// TIA Portal V20 export
FUNCTION_BLOCK "Sequence_10_GuageRnR"   // FB224, LAD
TITLE = Sequence
// Sequence template programmend in ladder logic
// stored: IsIECCheckEnabled true, MemoryReserve 100, Namespace Unit1.Em8, SetENOAutomatically true
   VAR_INPUT
      unitStatus { ExternalAccessible := 'False'; ExternalVisible := 'False'; ExternalWritable := 'False'} : "LAF_typeUnitStatus";
   END_VAR
   VAR
      instSequenceLADControl { ExternalAccessible := 'False'; ExternalVisible := 'False'; ExternalWritable := 'False'} : "LAF_ControlLadSequence";
      instSequenceLADStatus { ExternalAccessible := 'False'; ExternalVisible := 'False'; ExternalWritable := 'False'} : "LAF_StatusLadSequence";
      statTonTime { ExternalAccessible := 'False'; ExternalVisible := 'False'; ExternalWritable := 'False'} : Array[0..9999] of TON_TIME;
      NoDataCheck { S7_SetPoint := 'True'} : "LER_typePartData";
   END_VAR
   VAR_TEMP
      tempCustomerAction : Bool;   // Placeholder for possible actions
      tempDo_nothing_and_wait_for_init : Bool;   // Placeholder for doing nothing
      tempSafeStateCondition : Bool;   // Temp Condition for the equipment module to be in a safe state
   END_VAR
   VAR CONSTANT
      delayTime : Time := T#500ms;
      STEP_IDLE : DInt := 1;
      JOB_1_STEP_01 : DInt := 101;
      JOB_1_STEP_10 : DInt := 110;
      JOB_1_STEP_11 : DInt := 111;
      JOB_1_STEP_20 : DInt := 120;
      JOB_1_STEP_21 : DInt := 121;
      JOB_1_STEP_30 : DInt := 130;
      JOB_1_STEP_40 : DInt := 140;
      JOB_1_STEP_41 : DInt := 141;
      JOB_1_STEP_50 : DInt := 150;
      JOB_1_STEP_60 : DInt := 160;
      JOB_1_STEP_70 : DInt := 170;
      JOB_1_STEP_80 : DInt := 180;
      JOB_1_STEP_90 : DInt := 190;
      JOB_2_STEP_01 : DInt := 201;
      JOB_2_STEP_10 : DInt := 210;
      JOB_2_STEP_20 : DInt := 220;
      JOB_2_STEP_30 : DInt := 230;
      JOB_2_STEP_31 : DInt := 231;
      JOB_2_STEP_32 : DInt := 232;
      JOB_2_STEP_40 : DInt := 240;
      JOB_2_STEP_41 : DInt := 241;
      JOB_2_STEP_42 : DInt := 242;
      JOB_2_STEP_43 : DInt := 242;
      JOB_2_STEP_50 : DInt := 250;
      JOB_2_STEP_60 : DInt := 260;
      JOB_2_STEP_70 : DInt := 270;
      JOB_2_STEP_80 : DInt := 280;
      JOB_2_STEP_90 : DInt := 290;
      JOB_3_STEP_01 : DInt := 301;
      JOB_3_STEP_10 : DInt := 310;
      JOB_3_STEP_11 : DInt := 311;
      JOB_3_STEP_20 : DInt := 320;
      JOB_3_STEP_30 : DInt := 330;
      JOB_3_STEP_31 : DInt := 331;
      JOB_3_STEP_32 : DInt := 332;
      JOB_3_STEP_33 : DInt := 333;
      JOB_3_STEP_34 : DInt := 334;
      JOB_3_STEP_35 : DInt := 335;
      JOB_3_STEP_36 : DInt := 336;
      JOB_3_STEP_37 : DInt := 337;
      JOB_3_STEP_38 : DInt := 338;
      JOB_3_STEP_40 : DInt := 340;
      JOB_3_STEP_45 : DInt := 345;
      JOB_3_STEP_50 : DInt := 350;
      JOB_3_STEP_51 : DInt := 351;
      JOB_3_STEP_52 : DInt := 352;
      JOB_3_STEP_60 : DInt := 360;
      JOB_3_STEP_61 : DInt := 361;
      JOB_3_STEP_62 : DInt := 362;
      JOB_3_STEP_63 : DInt := 363;
      JOB_3_STEP_70 : DInt := 370;
      JOB_3_STEP_80 : DInt := 380;
      JOB_3_STEP_90 : DInt := 390;
      JOB_4_STEP_01 : DInt := 401;
      JOB_4_STEP_10 : DInt := 410;
      JOB_4_STEP_20 : DInt := 420;
      JOB_4_STEP_30 : DInt := 430;
      JOB_4_STEP_31 : DInt := 431;
      JOB_4_STEP_40 : DInt := 440;
      JOB_4_STEP_41 : DInt := 441;
      JOB_4_STEP_42 : DInt := 442;
      JOB_4_STEP_50 : DInt := 450;
      JOB_4_STEP_60 : DInt := 460;
      JOB_4_STEP_70 : DInt := 470;
      JOB_4_STEP_80 : DInt := 480;
      JOB_4_STEP_81 : DInt := 481;
      JOB_4_STEP_90 : DInt := 490;
      JOB_5_STEP_01 : DInt := 501;
      JOB_5_STEP_10 : DInt := 510;
      JOB_5_STEP_11 : DInt := 511;
      JOB_5_STEP_12 : DInt := 512;
      JOB_5_STEP_13 : DInt := 513;
      JOB_5_STEP_20 : DInt := 520;
      JOB_5_STEP_30 : DInt := 530;
      JOB_5_STEP_40 : DInt := 540;
      JOB_5_STEP_41 : DInt := 541;
      JOB_5_STEP_42 : DInt := 542;
      JOB_5_STEP_43 : DInt := 543;
      JOB_5_STEP_44 : DInt := 544;
      JOB_5_STEP_45 : DInt := 545;
      JOB_5_STEP_46 : DInt := 546;
      JOB_5_STEP_47 : DInt := 547;
      JOB_5_STEP_48 : DInt := 548;
      JOB_5_STEP_50 : DInt := 550;
      JOB_5_STEP_60 : DInt := 560;
      JOB_5_STEP_61 : DInt := 561;
      JOB_5_STEP_62 : DInt := 562;
      JOB_5_STEP_63 : DInt := 563;
      JOB_5_STEP_64 : DInt := 564;
      STEP_IMMEDIATE_STOP : DInt := 9001;   // Step executed when an immediate stop command is triggered for the sequence (i.e. when unit is in state aborting)
   END_VAR
   VAR_TEMP   // added for the SCL form of the ladder/FBD networks
      _w1 : Bool;
      _w2 : Bool;
      _w3 : Bool;
   END_VAR
BEGIN

REGION Network 1: BLOCK INFO HEADER
   // (company) / (C) Copyright (year)
   // ---------------------------------------------------------------------------------
   // Title:                             (Title of this block)
   // Comment/Function: (that is implemented in the block)
   // Library/Family:           (that the source is dedicated to)
   // Author:                        (department / person in charge / contact)
   // Target System:          (test system with FW version)
   // Engineering:              TIA Portal (SW version)
   // Restrictions:               (OB types, etc.)
   // Requirements:           (hardware, technological package, etc.)
   // ---------------------------------------------------------------------------------
   // Change log table:
   // Version          | Date             | Signature      | Expert in charge  | Changes applied ------------------------|----------------------|-------------------------|--------------------------------|-----------------------
   // 001.000.000 | yyyy-mm-dd | 0x00000000 | (name of expert) | First released version
END_REGION

REGION Network 2: DESCRIPTION
   // This is a template block provided by the Automation Framework. It can be used to create an own project.
   // The Block Info Header is prepared to put in your own data.
   // Description of the block could be added here and the docu created by Code2Docu.
END_REGION

REGION Network 3: ********************* CONTROL *************************
END_REGION

REGION Network 4: Sequence Control ("Enter your Sequins number here")
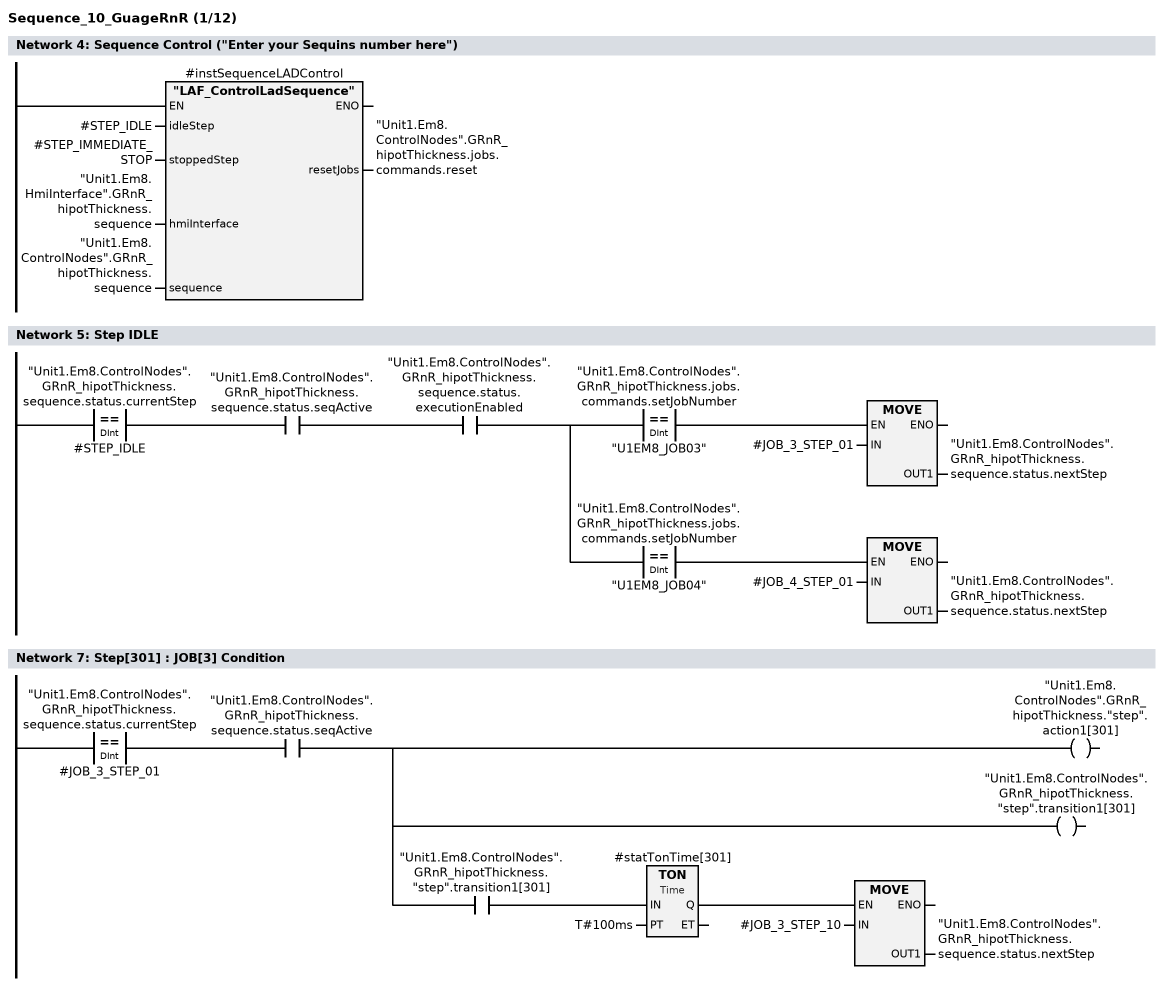
   RUNG wire#powerrail
      #instSequenceLADControl(idleStep := #STEP_IDLE, stoppedStep := #STEP_IMMEDIATE_STOP, hmiInterface := "Unit1.Em8.HmiInterface".GRnR_hipotThickness.sequence, sequence := "Unit1.Em8.ControlNodes".GRnR_hipotThickness.sequence, resetJobs => "Unit1.Em8.ControlNodes".GRnR_hipotThickness.jobs.commands.reset)
   END_RUNG
   // the same network as SCL:
   #instSequenceLADControl(idleStep := #STEP_IDLE,   // "LAF_ControlLadSequence"
                           stoppedStep := #STEP_IMMEDIATE_STOP,
                           hmiInterface := "Unit1.Em8.HmiInterface".GRnR_hipotThickness.sequence,
                           sequence := "Unit1.Em8.ControlNodes".GRnR_hipotThickness.sequence,
                           resetJobs => "Unit1.Em8.ControlNodes".GRnR_hipotThickness.jobs.commands.reset);
END_REGION

REGION Network 5: Step IDLE
   RUNG wire#powerrail
      { S7_Templates := "SrcType := DInt" } EQ_Contact(in1 := "Unit1.Em8.ControlNodes".GRnR_hipotThickness.sequence.status.currentStep, in2 := #STEP_IDLE)
      Contact( "Unit1.Em8.ControlNodes".GRnR_hipotThickness.sequence.status.seqActive )
      Contact( "Unit1.Em8.ControlNodes".GRnR_hipotThickness.sequence.status.executionEnabled )
      wire#w1
      { S7_Templates := "SrcType := DInt" } EQ_Contact(in1 := "Unit1.Em8.ControlNodes".GRnR_hipotThickness.jobs.commands.setJobNumber, in2 := "U1EM8_JOB03")
      Move(in := #JOB_3_STEP_01, out1 => "Unit1.Em8.ControlNodes".GRnR_hipotThickness.sequence.status.nextStep)
   END_RUNG
   RUNG wire#w1
      { S7_Templates := "SrcType := DInt" } EQ_Contact(in1 := "Unit1.Em8.ControlNodes".GRnR_hipotThickness.jobs.commands.setJobNumber, in2 := "U1EM8_JOB04")
      Move(in := #JOB_4_STEP_01, out1 => "Unit1.Em8.ControlNodes".GRnR_hipotThickness.sequence.status.nextStep)
   END_RUNG
   // the same network as SCL:
   #_w1 := ("Unit1.Em8.ControlNodes".GRnR_hipotThickness.sequence.status.currentStep = #STEP_IDLE) AND "Unit1.Em8.ControlNodes".GRnR_hipotThickness.sequence.status.seqActive AND "Unit1.Em8.ControlNodes".GRnR_hipotThickness.sequence.status.executionEnabled;
   IF #_w1 AND ("Unit1.Em8.ControlNodes".GRnR_hipotThickness.jobs.commands.setJobNumber = "U1EM8_JOB03") THEN
       "Unit1.Em8.ControlNodes".GRnR_hipotThickness.sequence.status.nextStep := #JOB_3_STEP_01;
   END_IF;
   IF #_w1 AND ("Unit1.Em8.ControlNodes".GRnR_hipotThickness.jobs.commands.setJobNumber = "U1EM8_JOB04") THEN
       "Unit1.Em8.ControlNodes".GRnR_hipotThickness.sequence.status.nextStep := #JOB_4_STEP_01;
   END_IF;
END_REGION

REGION Network 6: ************ JOB[3] JR HIPOT & THICKNESS=AUTO *************
END_REGION

REGION Network 7: Step[301] : JOB[3] Condition
   RUNG wire#powerrail
      { S7_Templates := "SrcType := DInt" } EQ_Contact(in1 := "Unit1.Em8.ControlNodes".GRnR_hipotThickness.sequence.status.currentStep, in2 := #JOB_3_STEP_01)
      Contact( "Unit1.Em8.ControlNodes".GRnR_hipotThickness.sequence.status.seqActive )
      wire#w1
      Coil( "Unit1.Em8.ControlNodes".GRnR_hipotThickness."step".action1[301] )
   END_RUNG
   RUNG wire#w1
      Coil( "Unit1.Em8.ControlNodes".GRnR_hipotThickness."step".transition1[301] )
   END_RUNG
   RUNG wire#w1
      Contact( "Unit1.Em8.ControlNodes".GRnR_hipotThickness."step".transition1[301] )
      { S7_Templates := "time_type := Time" } #statTonTime[301].TON(pt := T#100ms, et =>)
      Move(in := #JOB_3_STEP_10, out1 => "Unit1.Em8.ControlNodes".GRnR_hipotThickness.sequence.status.nextStep)
   END_RUNG
   // the same network as SCL:
   "Unit1.Em8.ControlNodes".GRnR_hipotThickness."step".action1[301] := ("Unit1.Em8.ControlNodes".GRnR_hipotThickness.sequence.status.currentStep = #JOB_3_STEP_01) AND "Unit1.Em8.ControlNodes".GRnR_hipotThickness.sequence.status.seqActive;
   "Unit1.Em8.ControlNodes".GRnR_hipotThickness."step".transition1[301] := ("Unit1.Em8.ControlNodes".GRnR_hipotThickness.sequence.status.currentStep = #JOB_3_STEP_01) AND "Unit1.Em8.ControlNodes".GRnR_hipotThickness.sequence.status.seqActive;
   #statTonTime[301].TON(IN := ("Unit1.Em8.ControlNodes".GRnR_hipotThickness.sequence.status.currentStep = #JOB_3_STEP_01) AND "Unit1.Em8.ControlNodes".GRnR_hipotThickness.sequence.status.seqActive AND "Unit1.Em8.ControlNodes".GRnR_hipotThickness."step".transition1[301],
                         PT := T#100ms);
   IF #statTonTime[301].Q THEN
       "Unit1.Em8.ControlNodes".GRnR_hipotThickness.sequence.status.nextStep := #JOB_3_STEP_10;
   END_IF;
END_REGION

REGION Network 8: Step[310] : Stage Lift Down
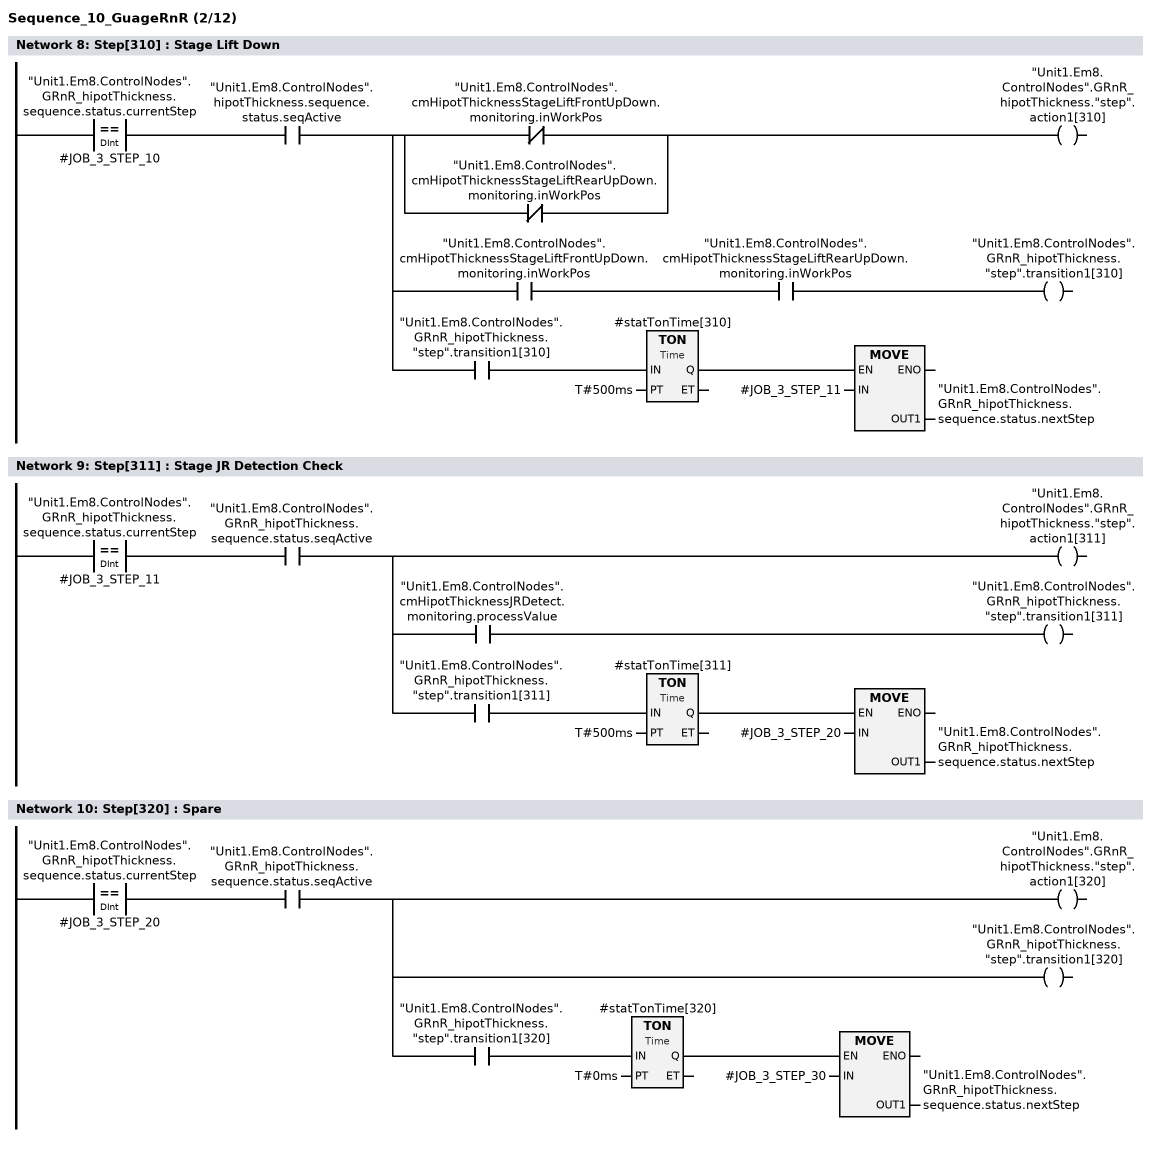
   RUNG wire#powerrail
      { S7_Templates := "SrcType := DInt" } EQ_Contact(in1 := "Unit1.Em8.ControlNodes".GRnR_hipotThickness.sequence.status.currentStep, in2 := #JOB_3_STEP_10)
      Contact( "Unit1.Em8.ControlNodes".hipotThickness.sequence.status.seqActive )
      wire#w1
      I_Contact( "Unit1.Em8.ControlNodes".cmHipotThicknessStageLiftFrontUpDown.monitoring.inWorkPos )
      wire#w2
      Coil( "Unit1.Em8.ControlNodes".GRnR_hipotThickness."step".action1[310] )
   END_RUNG
   RUNG wire#w1
      I_Contact( "Unit1.Em8.ControlNodes".cmHipotThicknessStageLiftRearUpDown.monitoring.inWorkPos )
   END_RUNG wire#w2
   RUNG wire#w1
      Contact( "Unit1.Em8.ControlNodes".cmHipotThicknessStageLiftFrontUpDown.monitoring.inWorkPos )
      Contact( "Unit1.Em8.ControlNodes".cmHipotThicknessStageLiftRearUpDown.monitoring.inWorkPos )
      Coil( "Unit1.Em8.ControlNodes".GRnR_hipotThickness."step".transition1[310] )
   END_RUNG
   RUNG wire#w1
      Contact( "Unit1.Em8.ControlNodes".GRnR_hipotThickness."step".transition1[310] )
      { S7_Templates := "time_type := Time" } #statTonTime[310].TON(pt := T#500ms, et =>)
      Move(in := #JOB_3_STEP_11, out1 => "Unit1.Em8.ControlNodes".GRnR_hipotThickness.sequence.status.nextStep)
   END_RUNG
   // the same network as SCL:
   #_w1 := ("Unit1.Em8.ControlNodes".GRnR_hipotThickness.sequence.status.currentStep = #JOB_3_STEP_10) AND "Unit1.Em8.ControlNodes".hipotThickness.sequence.status.seqActive;
   "Unit1.Em8.ControlNodes".GRnR_hipotThickness."step".action1[310] := #_w1 AND (NOT "Unit1.Em8.ControlNodes".cmHipotThicknessStageLiftFrontUpDown.monitoring.inWorkPos OR NOT "Unit1.Em8.ControlNodes".cmHipotThicknessStageLiftRearUpDown.monitoring.inWorkPos);
   "Unit1.Em8.ControlNodes".GRnR_hipotThickness."step".transition1[310] := #_w1 AND "Unit1.Em8.ControlNodes".cmHipotThicknessStageLiftFrontUpDown.monitoring.inWorkPos AND "Unit1.Em8.ControlNodes".cmHipotThicknessStageLiftRearUpDown.monitoring.inWorkPos;
   #statTonTime[310].TON(IN := #_w1 AND "Unit1.Em8.ControlNodes".GRnR_hipotThickness."step".transition1[310],
                         PT := T#500ms);
   IF #statTonTime[310].Q THEN
       "Unit1.Em8.ControlNodes".GRnR_hipotThickness.sequence.status.nextStep := #JOB_3_STEP_11;
   END_IF;
END_REGION

REGION Network 9: Step[311] : Stage JR Detection Check
   RUNG wire#powerrail
      { S7_Templates := "SrcType := DInt" } EQ_Contact(in1 := "Unit1.Em8.ControlNodes".GRnR_hipotThickness.sequence.status.currentStep, in2 := #JOB_3_STEP_11)
      Contact( "Unit1.Em8.ControlNodes".GRnR_hipotThickness.sequence.status.seqActive )
      wire#w1
      Coil( "Unit1.Em8.ControlNodes".GRnR_hipotThickness."step".action1[311] )
   END_RUNG
   RUNG wire#w1
      Contact( "Unit1.Em8.ControlNodes".cmHipotThicknessJRDetect.monitoring.processValue )
      Coil( "Unit1.Em8.ControlNodes".GRnR_hipotThickness."step".transition1[311] )
   END_RUNG
   RUNG wire#w1
      Contact( "Unit1.Em8.ControlNodes".GRnR_hipotThickness."step".transition1[311] )
      { S7_Templates := "time_type := Time" } #statTonTime[311].TON(pt := T#500ms, et =>)
      Move(in := #JOB_3_STEP_20, out1 => "Unit1.Em8.ControlNodes".GRnR_hipotThickness.sequence.status.nextStep)
   END_RUNG
   // the same network as SCL:
   "Unit1.Em8.ControlNodes".GRnR_hipotThickness."step".action1[311] := ("Unit1.Em8.ControlNodes".GRnR_hipotThickness.sequence.status.currentStep = #JOB_3_STEP_11) AND "Unit1.Em8.ControlNodes".GRnR_hipotThickness.sequence.status.seqActive;
   "Unit1.Em8.ControlNodes".GRnR_hipotThickness."step".transition1[311] := ("Unit1.Em8.ControlNodes".GRnR_hipotThickness.sequence.status.currentStep = #JOB_3_STEP_11) AND "Unit1.Em8.ControlNodes".GRnR_hipotThickness.sequence.status.seqActive AND "Unit1.Em8.ControlNodes".cmHipotThicknessJRDetect.monitoring.processValue;
   #statTonTime[311].TON(IN := ("Unit1.Em8.ControlNodes".GRnR_hipotThickness.sequence.status.currentStep = #JOB_3_STEP_11) AND "Unit1.Em8.ControlNodes".GRnR_hipotThickness.sequence.status.seqActive AND "Unit1.Em8.ControlNodes".GRnR_hipotThickness."step".transition1[311],
                         PT := T#500ms);
   IF #statTonTime[311].Q THEN
       "Unit1.Em8.ControlNodes".GRnR_hipotThickness.sequence.status.nextStep := #JOB_3_STEP_20;
   END_IF;
END_REGION

REGION Network 10: Step[320] : Spare
   RUNG wire#powerrail
      { S7_Templates := "SrcType := DInt" } EQ_Contact(in1 := "Unit1.Em8.ControlNodes".GRnR_hipotThickness.sequence.status.currentStep, in2 := #JOB_3_STEP_20)
      Contact( "Unit1.Em8.ControlNodes".GRnR_hipotThickness.sequence.status.seqActive )
      wire#w1
      Coil( "Unit1.Em8.ControlNodes".GRnR_hipotThickness."step".action1[320] )
   END_RUNG
   RUNG wire#w1
      Coil( "Unit1.Em8.ControlNodes".GRnR_hipotThickness."step".transition1[320] )
   END_RUNG
   RUNG wire#w1
      Contact( "Unit1.Em8.ControlNodes".GRnR_hipotThickness."step".transition1[320] )
      { S7_Templates := "time_type := Time" } #statTonTime[320].TON(pt := T#0ms, et =>)
      Move(in := #JOB_3_STEP_30, out1 => "Unit1.Em8.ControlNodes".GRnR_hipotThickness.sequence.status.nextStep)
   END_RUNG
   // the same network as SCL:
   "Unit1.Em8.ControlNodes".GRnR_hipotThickness."step".action1[320] := ("Unit1.Em8.ControlNodes".GRnR_hipotThickness.sequence.status.currentStep = #JOB_3_STEP_20) AND "Unit1.Em8.ControlNodes".GRnR_hipotThickness.sequence.status.seqActive;
   "Unit1.Em8.ControlNodes".GRnR_hipotThickness."step".transition1[320] := ("Unit1.Em8.ControlNodes".GRnR_hipotThickness.sequence.status.currentStep = #JOB_3_STEP_20) AND "Unit1.Em8.ControlNodes".GRnR_hipotThickness.sequence.status.seqActive;
   #statTonTime[320].TON(IN := ("Unit1.Em8.ControlNodes".GRnR_hipotThickness.sequence.status.currentStep = #JOB_3_STEP_20) AND "Unit1.Em8.ControlNodes".GRnR_hipotThickness.sequence.status.seqActive AND "Unit1.Em8.ControlNodes".GRnR_hipotThickness."step".transition1[320],
                         PT := T#0ms);
   IF #statTonTime[320].Q THEN
       "Unit1.Em8.ControlNodes".GRnR_hipotThickness.sequence.status.nextStep := #JOB_3_STEP_30;
   END_IF;
END_REGION

REGION Network 11: Step[330] : Press Start
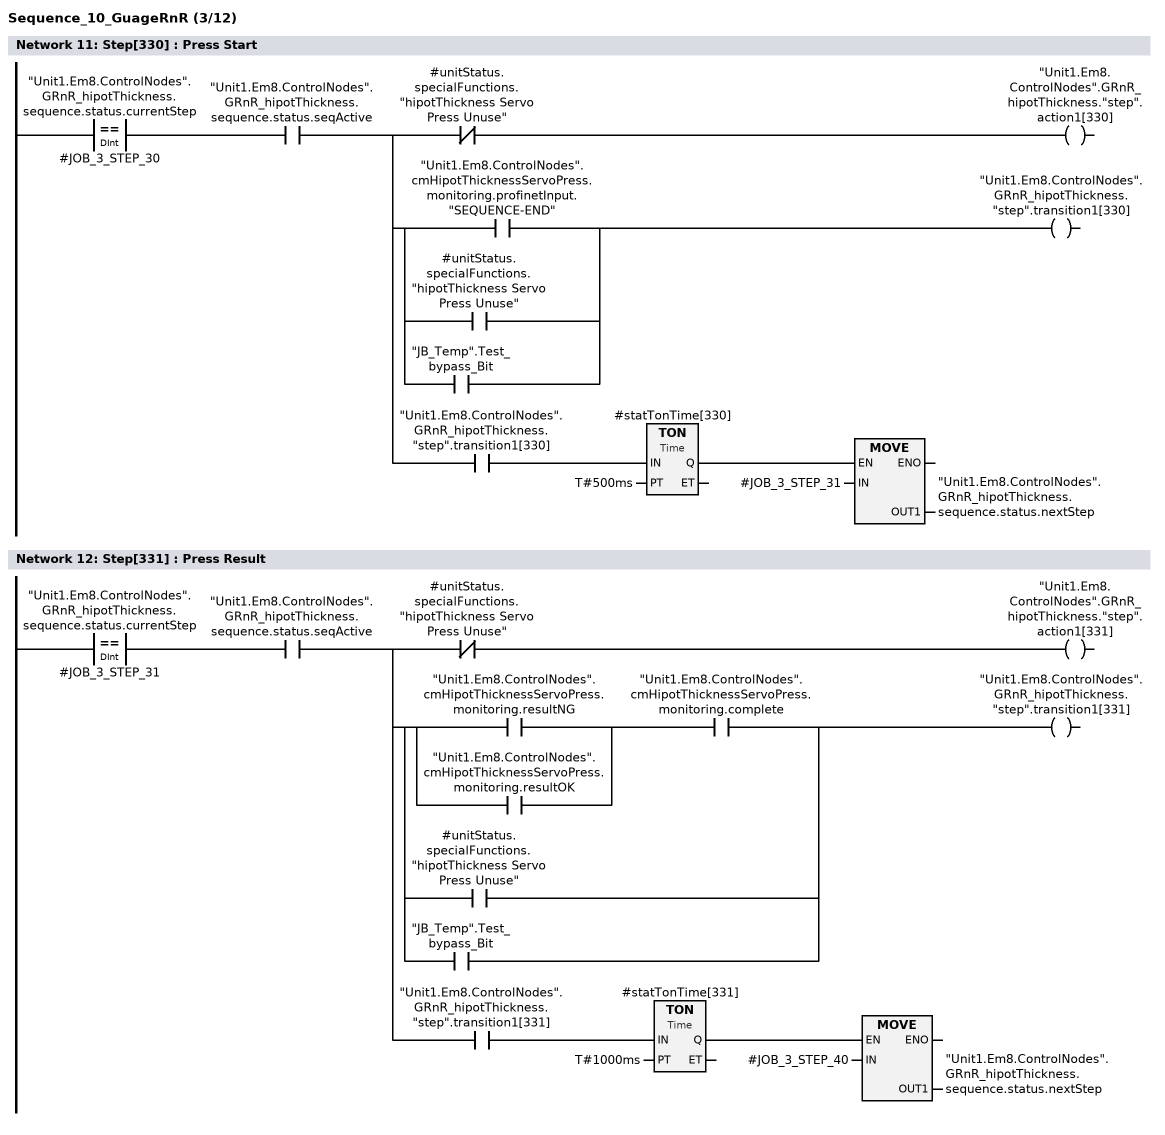
   RUNG wire#powerrail
      { S7_Templates := "SrcType := DInt" } EQ_Contact(in1 := "Unit1.Em8.ControlNodes".GRnR_hipotThickness.sequence.status.currentStep, in2 := #JOB_3_STEP_30)
      Contact( "Unit1.Em8.ControlNodes".GRnR_hipotThickness.sequence.status.seqActive )
      wire#w1
      I_Contact( #unitStatus.specialFunctions."hipotThickness Servo Press Unuse" )
      Coil( "Unit1.Em8.ControlNodes".GRnR_hipotThickness."step".action1[330] )
   END_RUNG
   RUNG wire#w1
      Contact( "Unit1.Em8.ControlNodes".cmHipotThicknessServoPress.monitoring.profinetInput."SEQUENCE-END" )
      wire#w2
      Coil( "Unit1.Em8.ControlNodes".GRnR_hipotThickness."step".transition1[330] )
   END_RUNG
   RUNG wire#w1
      Contact( #unitStatus.specialFunctions."hipotThickness Servo Press Unuse" )
   END_RUNG wire#w2
   RUNG wire#w1
      Contact( "JB_Temp".Test_bypass_Bit )
   END_RUNG wire#w2
   RUNG wire#w1
      Contact( "Unit1.Em8.ControlNodes".GRnR_hipotThickness."step".transition1[330] )
      { S7_Templates := "time_type := Time" } #statTonTime[330].TON(pt := T#500ms, et =>)
      Move(in := #JOB_3_STEP_31, out1 => "Unit1.Em8.ControlNodes".GRnR_hipotThickness.sequence.status.nextStep)
   END_RUNG
   // the same network as SCL:
   #_w1 := ("Unit1.Em8.ControlNodes".GRnR_hipotThickness.sequence.status.currentStep = #JOB_3_STEP_30) AND "Unit1.Em8.ControlNodes".GRnR_hipotThickness.sequence.status.seqActive;
   "Unit1.Em8.ControlNodes".GRnR_hipotThickness."step".action1[330] := #_w1 AND NOT #unitStatus.specialFunctions."hipotThickness Servo Press Unuse";
   "Unit1.Em8.ControlNodes".GRnR_hipotThickness."step".transition1[330] := #_w1 AND ("Unit1.Em8.ControlNodes".cmHipotThicknessServoPress.monitoring.profinetInput."SEQUENCE-END" OR #unitStatus.specialFunctions."hipotThickness Servo Press Unuse" OR "JB_Temp".Test_bypass_Bit);
   #statTonTime[330].TON(IN := #_w1 AND "Unit1.Em8.ControlNodes".GRnR_hipotThickness."step".transition1[330],
                         PT := T#500ms);
   IF #statTonTime[330].Q THEN
       "Unit1.Em8.ControlNodes".GRnR_hipotThickness.sequence.status.nextStep := #JOB_3_STEP_31;
   END_IF;
END_REGION

REGION Network 12: Step[331] : Press Result
   RUNG wire#powerrail
      { S7_Templates := "SrcType := DInt" } EQ_Contact(in1 := "Unit1.Em8.ControlNodes".GRnR_hipotThickness.sequence.status.currentStep, in2 := #JOB_3_STEP_31)
      Contact( "Unit1.Em8.ControlNodes".GRnR_hipotThickness.sequence.status.seqActive )
      wire#w1
      I_Contact( #unitStatus.specialFunctions."hipotThickness Servo Press Unuse" )
      Coil( "Unit1.Em8.ControlNodes".GRnR_hipotThickness."step".action1[331] )
   END_RUNG
   RUNG wire#w1
      Contact( "Unit1.Em8.ControlNodes".cmHipotThicknessServoPress.monitoring.resultNG )
      wire#w2
      Contact( "Unit1.Em8.ControlNodes".cmHipotThicknessServoPress.monitoring.complete )
      wire#w3
      Coil( "Unit1.Em8.ControlNodes".GRnR_hipotThickness."step".transition1[331] )
   END_RUNG
   RUNG wire#w1
      Contact( "Unit1.Em8.ControlNodes".cmHipotThicknessServoPress.monitoring.resultOK )
   END_RUNG wire#w2
   RUNG wire#w1
      Contact( #unitStatus.specialFunctions."hipotThickness Servo Press Unuse" )
   END_RUNG wire#w3
   RUNG wire#w1
      Contact( "JB_Temp".Test_bypass_Bit )
   END_RUNG wire#w3
   RUNG wire#w1
      Contact( "Unit1.Em8.ControlNodes".GRnR_hipotThickness."step".transition1[331] )
      { S7_Templates := "time_type := Time" } #statTonTime[331].TON(pt := T#1000ms, et =>)
      Move(in := #JOB_3_STEP_40, out1 => "Unit1.Em8.ControlNodes".GRnR_hipotThickness.sequence.status.nextStep)
   END_RUNG
   // the same network as SCL:
   #_w1 := ("Unit1.Em8.ControlNodes".GRnR_hipotThickness.sequence.status.currentStep = #JOB_3_STEP_31) AND "Unit1.Em8.ControlNodes".GRnR_hipotThickness.sequence.status.seqActive;
   "Unit1.Em8.ControlNodes".GRnR_hipotThickness."step".action1[331] := #_w1 AND NOT #unitStatus.specialFunctions."hipotThickness Servo Press Unuse";
   "Unit1.Em8.ControlNodes".GRnR_hipotThickness."step".transition1[331] := #_w1 AND ((("Unit1.Em8.ControlNodes".cmHipotThicknessServoPress.monitoring.resultNG OR "Unit1.Em8.ControlNodes".cmHipotThicknessServoPress.monitoring.resultOK) AND "Unit1.Em8.ControlNodes".cmHipotThicknessServoPress.monitoring.complete) OR #unitStatus.specialFunctions."hipotThickness Servo Press Unuse" OR "JB_Temp".Test_bypass_Bit);
   #statTonTime[331].TON(IN := #_w1 AND "Unit1.Em8.ControlNodes".GRnR_hipotThickness."step".transition1[331],
                         PT := T#1000ms);
   IF #statTonTime[331].Q THEN
       "Unit1.Em8.ControlNodes".GRnR_hipotThickness.sequence.status.nextStep := #JOB_3_STEP_40;
   END_IF;
END_REGION

REGION Network 13: Step[340] : Thickness Z-Axis Thickness Ready Pos, Tab Forward
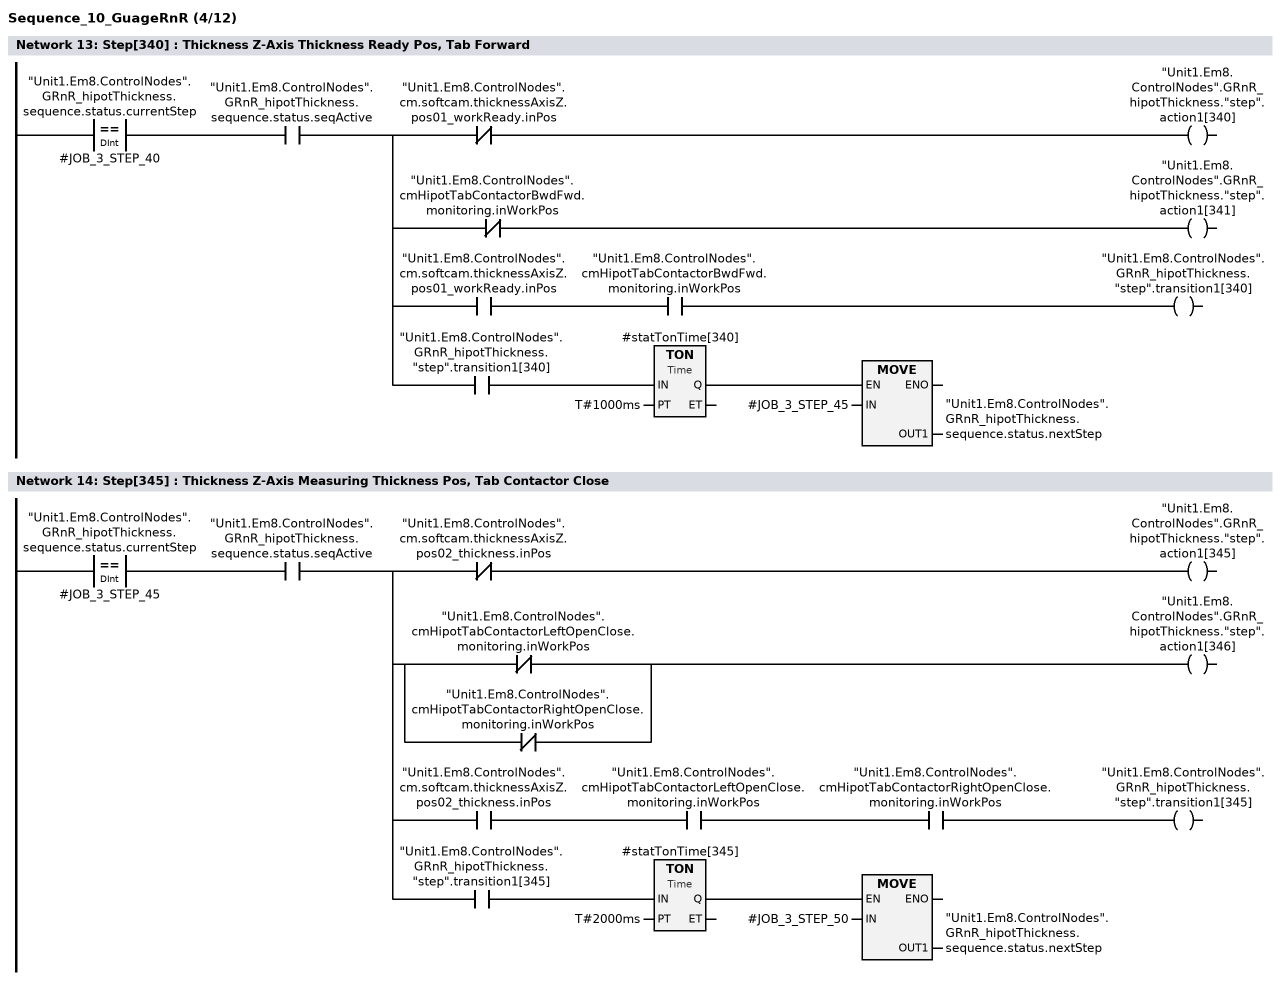
   RUNG wire#powerrail
      { S7_Templates := "SrcType := DInt" } EQ_Contact(in1 := "Unit1.Em8.ControlNodes".GRnR_hipotThickness.sequence.status.currentStep, in2 := #JOB_3_STEP_40)
      Contact( "Unit1.Em8.ControlNodes".GRnR_hipotThickness.sequence.status.seqActive )
      wire#w1
      I_Contact( "Unit1.Em8.ControlNodes".cm.softcam.thicknessAxisZ.pos01_workReady.inPos )
      Coil( "Unit1.Em8.ControlNodes".GRnR_hipotThickness."step".action1[340] )
   END_RUNG
   RUNG wire#w1
      I_Contact( "Unit1.Em8.ControlNodes".cmHipotTabContactorBwdFwd.monitoring.inWorkPos )
      Coil( "Unit1.Em8.ControlNodes".GRnR_hipotThickness."step".action1[341] )
   END_RUNG
   RUNG wire#w1
      Contact( "Unit1.Em8.ControlNodes".cm.softcam.thicknessAxisZ.pos01_workReady.inPos )
      Contact( "Unit1.Em8.ControlNodes".cmHipotTabContactorBwdFwd.monitoring.inWorkPos )
      Coil( "Unit1.Em8.ControlNodes".GRnR_hipotThickness."step".transition1[340] )
   END_RUNG
   RUNG wire#w1
      Contact( "Unit1.Em8.ControlNodes".GRnR_hipotThickness."step".transition1[340] )
      { S7_Templates := "time_type := Time" } #statTonTime[340].TON(pt := T#1000ms, et =>)
      Move(in := #JOB_3_STEP_45, out1 => "Unit1.Em8.ControlNodes".GRnR_hipotThickness.sequence.status.nextStep)
   END_RUNG
   // the same network as SCL:
   #_w1 := ("Unit1.Em8.ControlNodes".GRnR_hipotThickness.sequence.status.currentStep = #JOB_3_STEP_40) AND "Unit1.Em8.ControlNodes".GRnR_hipotThickness.sequence.status.seqActive;
   "Unit1.Em8.ControlNodes".GRnR_hipotThickness."step".action1[340] := #_w1 AND NOT "Unit1.Em8.ControlNodes".cm.softcam.thicknessAxisZ.pos01_workReady.inPos;
   "Unit1.Em8.ControlNodes".GRnR_hipotThickness."step".action1[341] := #_w1 AND NOT "Unit1.Em8.ControlNodes".cmHipotTabContactorBwdFwd.monitoring.inWorkPos;
   "Unit1.Em8.ControlNodes".GRnR_hipotThickness."step".transition1[340] := #_w1 AND "Unit1.Em8.ControlNodes".cm.softcam.thicknessAxisZ.pos01_workReady.inPos AND "Unit1.Em8.ControlNodes".cmHipotTabContactorBwdFwd.monitoring.inWorkPos;
   #statTonTime[340].TON(IN := #_w1 AND "Unit1.Em8.ControlNodes".GRnR_hipotThickness."step".transition1[340],
                         PT := T#1000ms);
   IF #statTonTime[340].Q THEN
       "Unit1.Em8.ControlNodes".GRnR_hipotThickness.sequence.status.nextStep := #JOB_3_STEP_45;
   END_IF;
END_REGION

REGION Network 14: Step[345] : Thickness Z-Axis Measuring Thickness Pos, Tab Contactor Close
   RUNG wire#powerrail
      { S7_Templates := "SrcType := DInt" } EQ_Contact(in1 := "Unit1.Em8.ControlNodes".GRnR_hipotThickness.sequence.status.currentStep, in2 := #JOB_3_STEP_45)
      Contact( "Unit1.Em8.ControlNodes".GRnR_hipotThickness.sequence.status.seqActive )
      wire#w1
      I_Contact( "Unit1.Em8.ControlNodes".cm.softcam.thicknessAxisZ.pos02_thickness.inPos )
      Coil( "Unit1.Em8.ControlNodes".GRnR_hipotThickness."step".action1[345] )
   END_RUNG
   RUNG wire#w1
      I_Contact( "Unit1.Em8.ControlNodes".cmHipotTabContactorLeftOpenClose.monitoring.inWorkPos )
      wire#w2
      Coil( "Unit1.Em8.ControlNodes".GRnR_hipotThickness."step".action1[346] )
   END_RUNG
   RUNG wire#w1
      I_Contact( "Unit1.Em8.ControlNodes".cmHipotTabContactorRightOpenClose.monitoring.inWorkPos )
   END_RUNG wire#w2
   RUNG wire#w1
      Contact( "Unit1.Em8.ControlNodes".cm.softcam.thicknessAxisZ.pos02_thickness.inPos )
      Contact( "Unit1.Em8.ControlNodes".cmHipotTabContactorLeftOpenClose.monitoring.inWorkPos )
      Contact( "Unit1.Em8.ControlNodes".cmHipotTabContactorRightOpenClose.monitoring.inWorkPos )
      Coil( "Unit1.Em8.ControlNodes".GRnR_hipotThickness."step".transition1[345] )
   END_RUNG
   RUNG wire#w1
      Contact( "Unit1.Em8.ControlNodes".GRnR_hipotThickness."step".transition1[345] )
      { S7_Templates := "time_type := Time" } #statTonTime[345].TON(pt := T#2000ms, et =>)
      Move(in := #JOB_3_STEP_50, out1 => "Unit1.Em8.ControlNodes".GRnR_hipotThickness.sequence.status.nextStep)
   END_RUNG
   // the same network as SCL:
   #_w1 := ("Unit1.Em8.ControlNodes".GRnR_hipotThickness.sequence.status.currentStep = #JOB_3_STEP_45) AND "Unit1.Em8.ControlNodes".GRnR_hipotThickness.sequence.status.seqActive;
   "Unit1.Em8.ControlNodes".GRnR_hipotThickness."step".action1[345] := #_w1 AND NOT "Unit1.Em8.ControlNodes".cm.softcam.thicknessAxisZ.pos02_thickness.inPos;
   "Unit1.Em8.ControlNodes".GRnR_hipotThickness."step".action1[346] := #_w1 AND (NOT "Unit1.Em8.ControlNodes".cmHipotTabContactorLeftOpenClose.monitoring.inWorkPos OR NOT "Unit1.Em8.ControlNodes".cmHipotTabContactorRightOpenClose.monitoring.inWorkPos);
   "Unit1.Em8.ControlNodes".GRnR_hipotThickness."step".transition1[345] := #_w1 AND "Unit1.Em8.ControlNodes".cm.softcam.thicknessAxisZ.pos02_thickness.inPos AND "Unit1.Em8.ControlNodes".cmHipotTabContactorLeftOpenClose.monitoring.inWorkPos AND "Unit1.Em8.ControlNodes".cmHipotTabContactorRightOpenClose.monitoring.inWorkPos;
   #statTonTime[345].TON(IN := #_w1 AND "Unit1.Em8.ControlNodes".GRnR_hipotThickness."step".transition1[345],
                         PT := T#2000ms);
   IF #statTonTime[345].Q THEN
       "Unit1.Em8.ControlNodes".GRnR_hipotThickness.sequence.status.nextStep := #JOB_3_STEP_50;
   END_IF;
END_REGION

REGION Network 15: Step[350] : Thickness Start
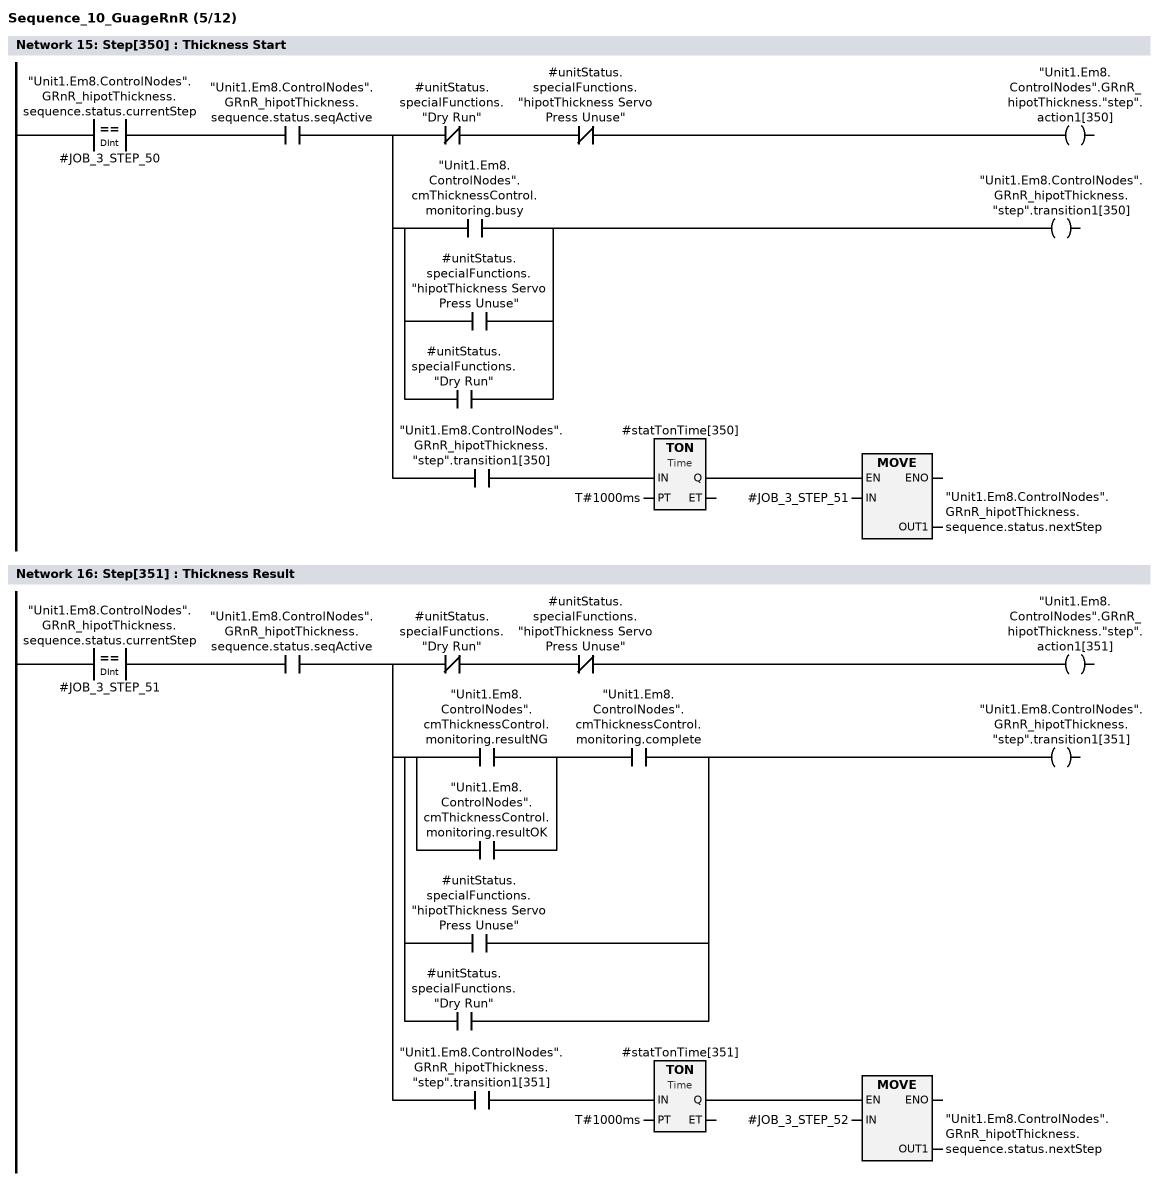
   RUNG wire#powerrail
      { S7_Templates := "SrcType := DInt" } EQ_Contact(in1 := "Unit1.Em8.ControlNodes".GRnR_hipotThickness.sequence.status.currentStep, in2 := #JOB_3_STEP_50)
      Contact( "Unit1.Em8.ControlNodes".GRnR_hipotThickness.sequence.status.seqActive )
      wire#w1
      I_Contact( #unitStatus.specialFunctions."Dry Run" )
      I_Contact( #unitStatus.specialFunctions."hipotThickness Servo Press Unuse" )
      Coil( "Unit1.Em8.ControlNodes".GRnR_hipotThickness."step".action1[350] )
   END_RUNG
   RUNG wire#w1
      Contact( "Unit1.Em8.ControlNodes".cmThicknessControl.monitoring.busy )
      wire#w2
      Coil( "Unit1.Em8.ControlNodes".GRnR_hipotThickness."step".transition1[350] )
   END_RUNG
   RUNG wire#w1
      Contact( #unitStatus.specialFunctions."hipotThickness Servo Press Unuse" )
   END_RUNG wire#w2
   RUNG wire#w1
      Contact( #unitStatus.specialFunctions."Dry Run" )
   END_RUNG wire#w2
   RUNG wire#w1
      Contact( "Unit1.Em8.ControlNodes".GRnR_hipotThickness."step".transition1[350] )
      { S7_Templates := "time_type := Time" } #statTonTime[350].TON(pt := T#1000ms, et =>)
      Move(in := #JOB_3_STEP_51, out1 => "Unit1.Em8.ControlNodes".GRnR_hipotThickness.sequence.status.nextStep)
   END_RUNG
   // the same network as SCL:
   #_w1 := ("Unit1.Em8.ControlNodes".GRnR_hipotThickness.sequence.status.currentStep = #JOB_3_STEP_50) AND "Unit1.Em8.ControlNodes".GRnR_hipotThickness.sequence.status.seqActive;
   "Unit1.Em8.ControlNodes".GRnR_hipotThickness."step".action1[350] := #_w1 AND NOT #unitStatus.specialFunctions."Dry Run" AND NOT #unitStatus.specialFunctions."hipotThickness Servo Press Unuse";
   "Unit1.Em8.ControlNodes".GRnR_hipotThickness."step".transition1[350] := #_w1 AND ("Unit1.Em8.ControlNodes".cmThicknessControl.monitoring.busy OR #unitStatus.specialFunctions."hipotThickness Servo Press Unuse" OR #unitStatus.specialFunctions."Dry Run");
   #statTonTime[350].TON(IN := #_w1 AND "Unit1.Em8.ControlNodes".GRnR_hipotThickness."step".transition1[350],
                         PT := T#1000ms);
   IF #statTonTime[350].Q THEN
       "Unit1.Em8.ControlNodes".GRnR_hipotThickness.sequence.status.nextStep := #JOB_3_STEP_51;
   END_IF;
END_REGION

REGION Network 16: Step[351] : Thickness Result
   RUNG wire#powerrail
      { S7_Templates := "SrcType := DInt" } EQ_Contact(in1 := "Unit1.Em8.ControlNodes".GRnR_hipotThickness.sequence.status.currentStep, in2 := #JOB_3_STEP_51)
      Contact( "Unit1.Em8.ControlNodes".GRnR_hipotThickness.sequence.status.seqActive )
      wire#w1
      I_Contact( #unitStatus.specialFunctions."Dry Run" )
      I_Contact( #unitStatus.specialFunctions."hipotThickness Servo Press Unuse" )
      Coil( "Unit1.Em8.ControlNodes".GRnR_hipotThickness."step".action1[351] )
   END_RUNG
   RUNG wire#w1
      Contact( "Unit1.Em8.ControlNodes".cmThicknessControl.monitoring.resultNG )
      wire#w2
      Contact( "Unit1.Em8.ControlNodes".cmThicknessControl.monitoring.complete )
      wire#w3
      Coil( "Unit1.Em8.ControlNodes".GRnR_hipotThickness."step".transition1[351] )
   END_RUNG
   RUNG wire#w1
      Contact( "Unit1.Em8.ControlNodes".cmThicknessControl.monitoring.resultOK )
   END_RUNG wire#w2
   RUNG wire#w1
      Contact( #unitStatus.specialFunctions."hipotThickness Servo Press Unuse" )
   END_RUNG wire#w3
   RUNG wire#w1
      Contact( #unitStatus.specialFunctions."Dry Run" )
   END_RUNG wire#w3
   RUNG wire#w1
      Contact( "Unit1.Em8.ControlNodes".GRnR_hipotThickness."step".transition1[351] )
      { S7_Templates := "time_type := Time" } #statTonTime[351].TON(pt := T#1000ms, et =>)
      Move(in := #JOB_3_STEP_52, out1 => "Unit1.Em8.ControlNodes".GRnR_hipotThickness.sequence.status.nextStep)
   END_RUNG
   // the same network as SCL:
   #_w1 := ("Unit1.Em8.ControlNodes".GRnR_hipotThickness.sequence.status.currentStep = #JOB_3_STEP_51) AND "Unit1.Em8.ControlNodes".GRnR_hipotThickness.sequence.status.seqActive;
   "Unit1.Em8.ControlNodes".GRnR_hipotThickness."step".action1[351] := #_w1 AND NOT #unitStatus.specialFunctions."Dry Run" AND NOT #unitStatus.specialFunctions."hipotThickness Servo Press Unuse";
   "Unit1.Em8.ControlNodes".GRnR_hipotThickness."step".transition1[351] := #_w1 AND ((("Unit1.Em8.ControlNodes".cmThicknessControl.monitoring.resultNG OR "Unit1.Em8.ControlNodes".cmThicknessControl.monitoring.resultOK) AND "Unit1.Em8.ControlNodes".cmThicknessControl.monitoring.complete) OR #unitStatus.specialFunctions."hipotThickness Servo Press Unuse" OR #unitStatus.specialFunctions."Dry Run");
   #statTonTime[351].TON(IN := #_w1 AND "Unit1.Em8.ControlNodes".GRnR_hipotThickness."step".transition1[351],
                         PT := T#1000ms);
   IF #statTonTime[351].Q THEN
       "Unit1.Em8.ControlNodes".GRnR_hipotThickness.sequence.status.nextStep := #JOB_3_STEP_52;
   END_IF;
END_REGION

REGION Network 17: Step[352] : Thickness Z-Axis Wait Pos
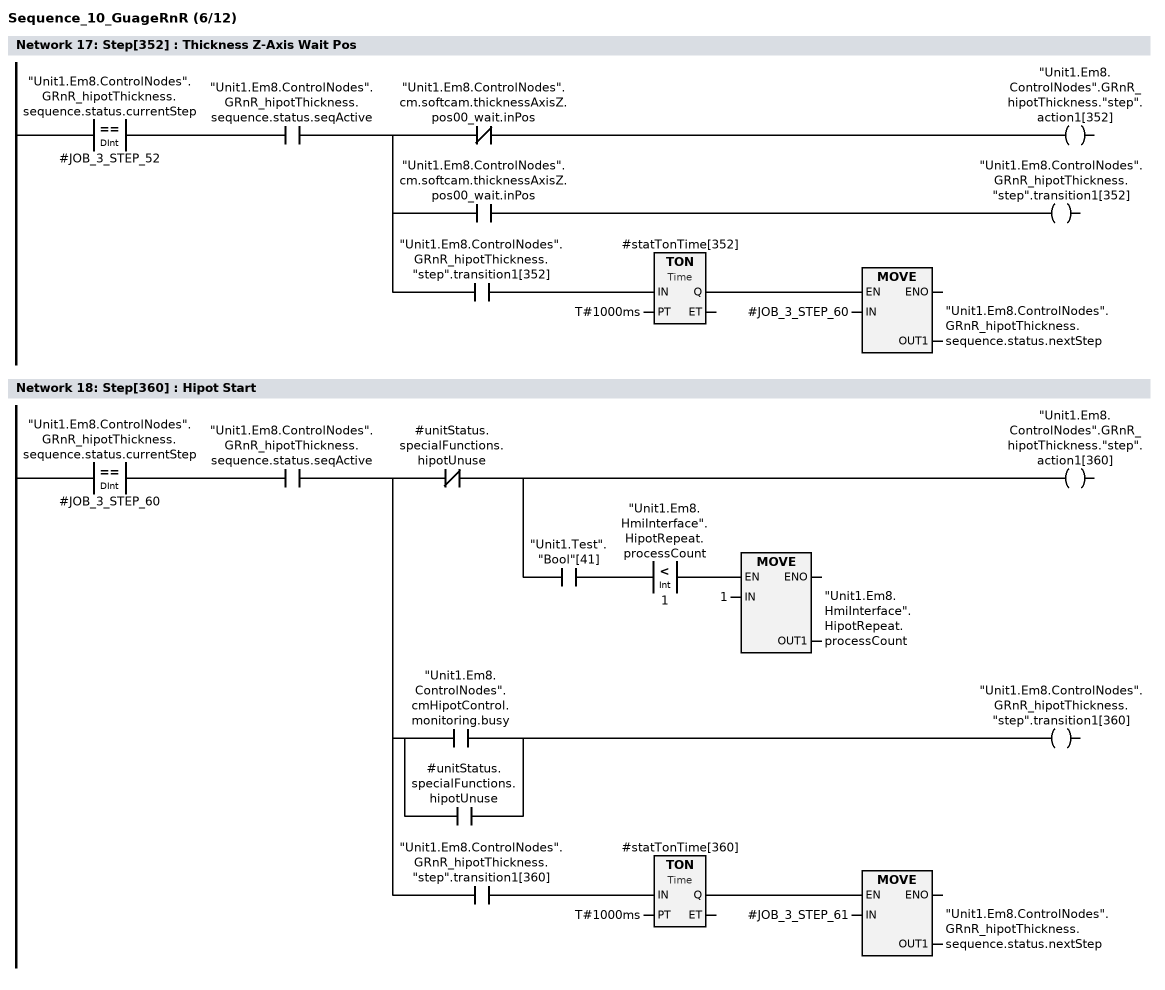
   RUNG wire#powerrail
      { S7_Templates := "SrcType := DInt" } EQ_Contact(in1 := "Unit1.Em8.ControlNodes".GRnR_hipotThickness.sequence.status.currentStep, in2 := #JOB_3_STEP_52)
      Contact( "Unit1.Em8.ControlNodes".GRnR_hipotThickness.sequence.status.seqActive )
      wire#w1
      I_Contact( "Unit1.Em8.ControlNodes".cm.softcam.thicknessAxisZ.pos00_wait.inPos )
      Coil( "Unit1.Em8.ControlNodes".GRnR_hipotThickness."step".action1[352] )
   END_RUNG
   RUNG wire#w1
      Contact( "Unit1.Em8.ControlNodes".cm.softcam.thicknessAxisZ.pos00_wait.inPos )
      Coil( "Unit1.Em8.ControlNodes".GRnR_hipotThickness."step".transition1[352] )
   END_RUNG
   RUNG wire#w1
      Contact( "Unit1.Em8.ControlNodes".GRnR_hipotThickness."step".transition1[352] )
      { S7_Templates := "time_type := Time" } #statTonTime[352].TON(pt := T#1000ms, et =>)
      Move(in := #JOB_3_STEP_60, out1 => "Unit1.Em8.ControlNodes".GRnR_hipotThickness.sequence.status.nextStep)
   END_RUNG
   // the same network as SCL:
   #_w1 := ("Unit1.Em8.ControlNodes".GRnR_hipotThickness.sequence.status.currentStep = #JOB_3_STEP_52) AND "Unit1.Em8.ControlNodes".GRnR_hipotThickness.sequence.status.seqActive;
   "Unit1.Em8.ControlNodes".GRnR_hipotThickness."step".action1[352] := #_w1 AND NOT "Unit1.Em8.ControlNodes".cm.softcam.thicknessAxisZ.pos00_wait.inPos;
   "Unit1.Em8.ControlNodes".GRnR_hipotThickness."step".transition1[352] := #_w1 AND "Unit1.Em8.ControlNodes".cm.softcam.thicknessAxisZ.pos00_wait.inPos;
   #statTonTime[352].TON(IN := #_w1 AND "Unit1.Em8.ControlNodes".GRnR_hipotThickness."step".transition1[352],
                         PT := T#1000ms);
   IF #statTonTime[352].Q THEN
       "Unit1.Em8.ControlNodes".GRnR_hipotThickness.sequence.status.nextStep := #JOB_3_STEP_60;
   END_IF;
END_REGION

REGION Network 18: Step[360] : Hipot Start
   RUNG wire#powerrail
      { S7_Templates := "SrcType := DInt" } EQ_Contact(in1 := "Unit1.Em8.ControlNodes".GRnR_hipotThickness.sequence.status.currentStep, in2 := #JOB_3_STEP_60)
      Contact( "Unit1.Em8.ControlNodes".GRnR_hipotThickness.sequence.status.seqActive )
      wire#w1
      I_Contact( #unitStatus.specialFunctions.hipotUnuse )
      wire#w2
      Coil( "Unit1.Em8.ControlNodes".GRnR_hipotThickness."step".action1[360] )
   END_RUNG
   RUNG wire#w2
      Contact( "Unit1.Test"."Bool"[41] )
      { S7_Templates := "SrcType := Int" } LT_Contact(in1 := "Unit1.Em8.HmiInterface".HipotRepeat.processCount, in2 := 1)
      Move(in := 1, out1 => "Unit1.Em8.HmiInterface".HipotRepeat.processCount)
   END_RUNG
   RUNG wire#w1
      Contact( "Unit1.Em8.ControlNodes".cmHipotControl.monitoring.busy )
      wire#w3
      Coil( "Unit1.Em8.ControlNodes".GRnR_hipotThickness."step".transition1[360] )
   END_RUNG
   RUNG wire#w1
      Contact( #unitStatus.specialFunctions.hipotUnuse )
   END_RUNG wire#w3
   RUNG wire#w1
      Contact( "Unit1.Em8.ControlNodes".GRnR_hipotThickness."step".transition1[360] )
      { S7_Templates := "time_type := Time" } #statTonTime[360].TON(pt := T#1000ms, et =>)
      Move(in := #JOB_3_STEP_61, out1 => "Unit1.Em8.ControlNodes".GRnR_hipotThickness.sequence.status.nextStep)
   END_RUNG
   // the same network as SCL:
   #_w1 := ("Unit1.Em8.ControlNodes".GRnR_hipotThickness.sequence.status.currentStep = #JOB_3_STEP_60) AND "Unit1.Em8.ControlNodes".GRnR_hipotThickness.sequence.status.seqActive;
   "Unit1.Em8.ControlNodes".GRnR_hipotThickness."step".action1[360] := #_w1 AND NOT #unitStatus.specialFunctions.hipotUnuse;
   IF #_w1 AND NOT #unitStatus.specialFunctions.hipotUnuse AND "Unit1.Test"."Bool"[41] AND ("Unit1.Em8.HmiInterface".HipotRepeat.processCount < 1) THEN
       "Unit1.Em8.HmiInterface".HipotRepeat.processCount := 1;
   END_IF;
   "Unit1.Em8.ControlNodes".GRnR_hipotThickness."step".transition1[360] := #_w1 AND ("Unit1.Em8.ControlNodes".cmHipotControl.monitoring.busy OR #unitStatus.specialFunctions.hipotUnuse);
   #statTonTime[360].TON(IN := #_w1 AND "Unit1.Em8.ControlNodes".GRnR_hipotThickness."step".transition1[360],
                         PT := T#1000ms);
   IF #statTonTime[360].Q THEN
       "Unit1.Em8.ControlNodes".GRnR_hipotThickness.sequence.status.nextStep := #JOB_3_STEP_61;
   END_IF;
END_REGION

REGION Network 19: Step[361] : Hipot Result
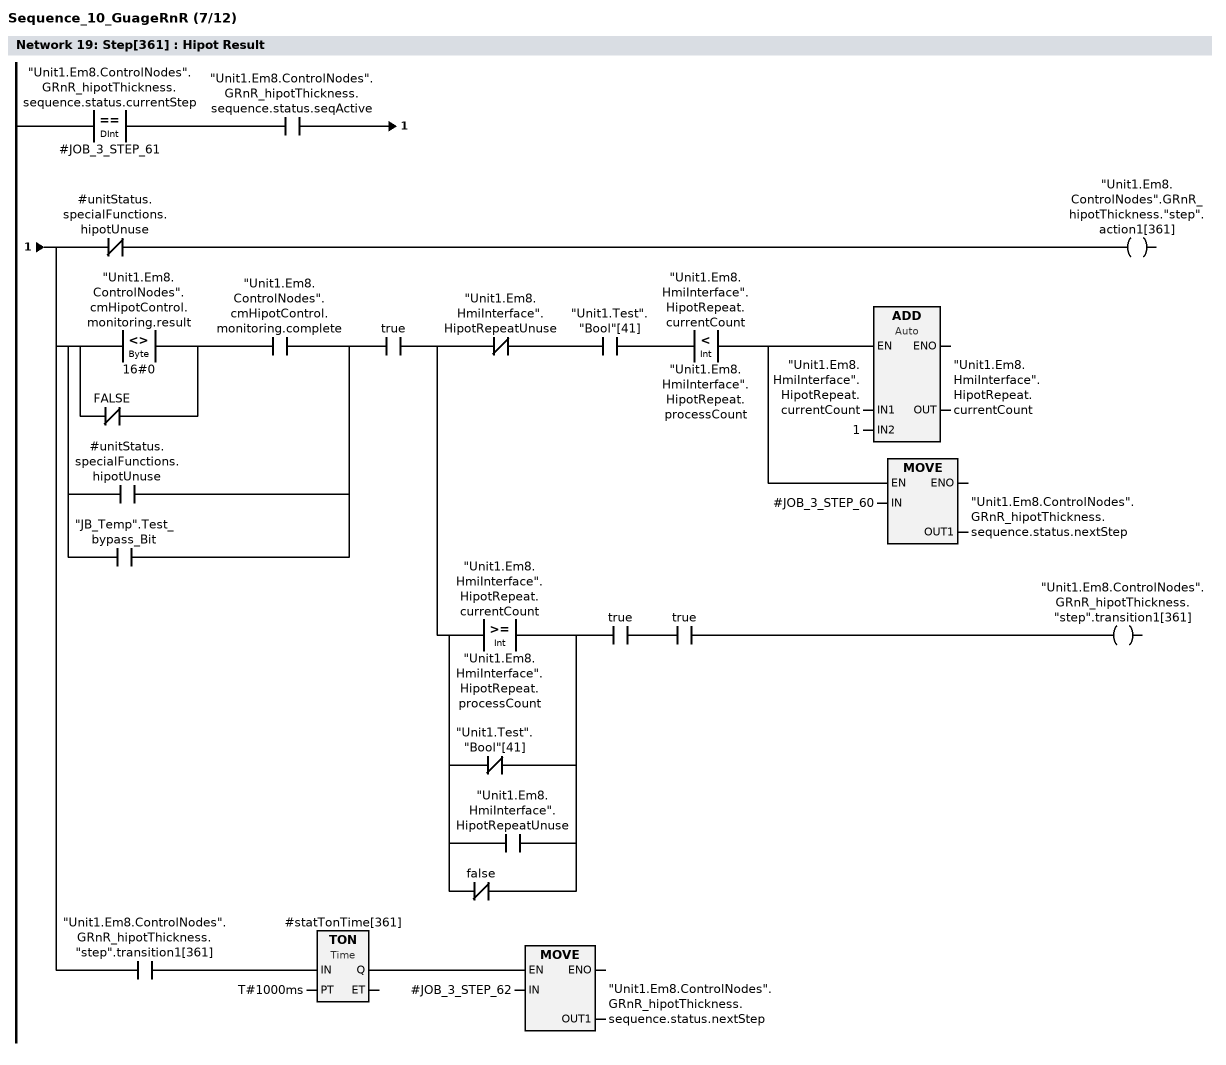
   RUNG wire#powerrail
      { S7_Templates := "SrcType := DInt" } EQ_Contact(in1 := "Unit1.Em8.ControlNodes".GRnR_hipotThickness.sequence.status.currentStep, in2 := #JOB_3_STEP_61)
      Contact( "Unit1.Em8.ControlNodes".GRnR_hipotThickness.sequence.status.seqActive )
      wire#w1
      I_Contact( #unitStatus.specialFunctions.hipotUnuse )
      Coil( "Unit1.Em8.ControlNodes".GRnR_hipotThickness."step".action1[361] )
   END_RUNG
   RUNG wire#w1
      { S7_Templates := "SrcType := Byte" } NE_Contact(in1 := "Unit1.Em8.ControlNodes".cmHipotControl.monitoring.result, in2 := 16#0)
      wire#w2
      Contact( "Unit1.Em8.ControlNodes".cmHipotControl.monitoring.complete )
      wire#w3
      Contact( true )
      wire#w4
      I_Contact( "Unit1.Em8.HmiInterface".HipotRepeatUnuse )
      Contact( "Unit1.Test"."Bool"[41] )
      { S7_Templates := "SrcType := Int" } LT_Contact(in1 := "Unit1.Em8.HmiInterface".HipotRepeat.currentCount, in2 := "Unit1.Em8.HmiInterface".HipotRepeat.processCount)
      wire#w5
      Add(in1 := "Unit1.Em8.HmiInterface".HipotRepeat.currentCount, in2 := 1, out => "Unit1.Em8.HmiInterface".HipotRepeat.currentCount)
   END_RUNG
   RUNG wire#w1
      I_Contact( FALSE )
   END_RUNG wire#w2
   RUNG wire#w1
      Contact( #unitStatus.specialFunctions.hipotUnuse )
   END_RUNG wire#w3
   RUNG wire#w1
      Contact( "JB_Temp".Test_bypass_Bit )
   END_RUNG wire#w3
   RUNG wire#w5
      Move(in := #JOB_3_STEP_60, out1 => "Unit1.Em8.ControlNodes".GRnR_hipotThickness.sequence.status.nextStep)
   END_RUNG
   RUNG wire#w4
      { S7_Templates := "SrcType := Int" } GE_Contact(in1 := "Unit1.Em8.HmiInterface".HipotRepeat.currentCount, in2 := "Unit1.Em8.HmiInterface".HipotRepeat.processCount)
      wire#w6
      Contact( true )
      Contact( true )
      Coil( "Unit1.Em8.ControlNodes".GRnR_hipotThickness."step".transition1[361] )
   END_RUNG
   RUNG wire#w4
      I_Contact( "Unit1.Test"."Bool"[41] )
   END_RUNG wire#w6
   RUNG wire#w4
      Contact( "Unit1.Em8.HmiInterface".HipotRepeatUnuse )
   END_RUNG wire#w6
   RUNG wire#w4
      I_Contact( false )
   END_RUNG wire#w6
   RUNG wire#w1
      Contact( "Unit1.Em8.ControlNodes".GRnR_hipotThickness."step".transition1[361] )
      { S7_Templates := "time_type := Time" } #statTonTime[361].TON(pt := T#1000ms, et =>)
      Move(in := #JOB_3_STEP_62, out1 => "Unit1.Em8.ControlNodes".GRnR_hipotThickness.sequence.status.nextStep)
   END_RUNG
   // the same network as SCL:
   #_w1 := ("Unit1.Em8.ControlNodes".GRnR_hipotThickness.sequence.status.currentStep = #JOB_3_STEP_61) AND "Unit1.Em8.ControlNodes".GRnR_hipotThickness.sequence.status.seqActive;
   "Unit1.Em8.ControlNodes".GRnR_hipotThickness."step".action1[361] := #_w1 AND NOT #unitStatus.specialFunctions.hipotUnuse;
   #_w2 := #_w1 AND (((("Unit1.Em8.ControlNodes".cmHipotControl.monitoring.result <> 16#0) OR NOT FALSE) AND "Unit1.Em8.ControlNodes".cmHipotControl.monitoring.complete) OR #unitStatus.specialFunctions.hipotUnuse OR "JB_Temp".Test_bypass_Bit) AND true;
   #_w3 := #_w2 AND NOT "Unit1.Em8.HmiInterface".HipotRepeatUnuse AND "Unit1.Test"."Bool"[41] AND ("Unit1.Em8.HmiInterface".HipotRepeat.currentCount < "Unit1.Em8.HmiInterface".HipotRepeat.processCount);
   IF #_w3 THEN
       "Unit1.Em8.HmiInterface".HipotRepeat.currentCount := "Unit1.Em8.HmiInterface".HipotRepeat.currentCount + 1;
       "Unit1.Em8.ControlNodes".GRnR_hipotThickness.sequence.status.nextStep := #JOB_3_STEP_60;
   END_IF;
   "Unit1.Em8.ControlNodes".GRnR_hipotThickness."step".transition1[361] := #_w2 AND (("Unit1.Em8.HmiInterface".HipotRepeat.currentCount >= "Unit1.Em8.HmiInterface".HipotRepeat.processCount) OR NOT "Unit1.Test"."Bool"[41] OR "Unit1.Em8.HmiInterface".HipotRepeatUnuse OR NOT false) AND true AND true;
   #statTonTime[361].TON(IN := #_w1 AND "Unit1.Em8.ControlNodes".GRnR_hipotThickness."step".transition1[361],
                         PT := T#1000ms);
   IF #statTonTime[361].Q THEN
       "Unit1.Em8.ControlNodes".GRnR_hipotThickness.sequence.status.nextStep := #JOB_3_STEP_62;
   END_IF;
END_REGION

REGION Network 20: Step[362] : Tab Contactor Open
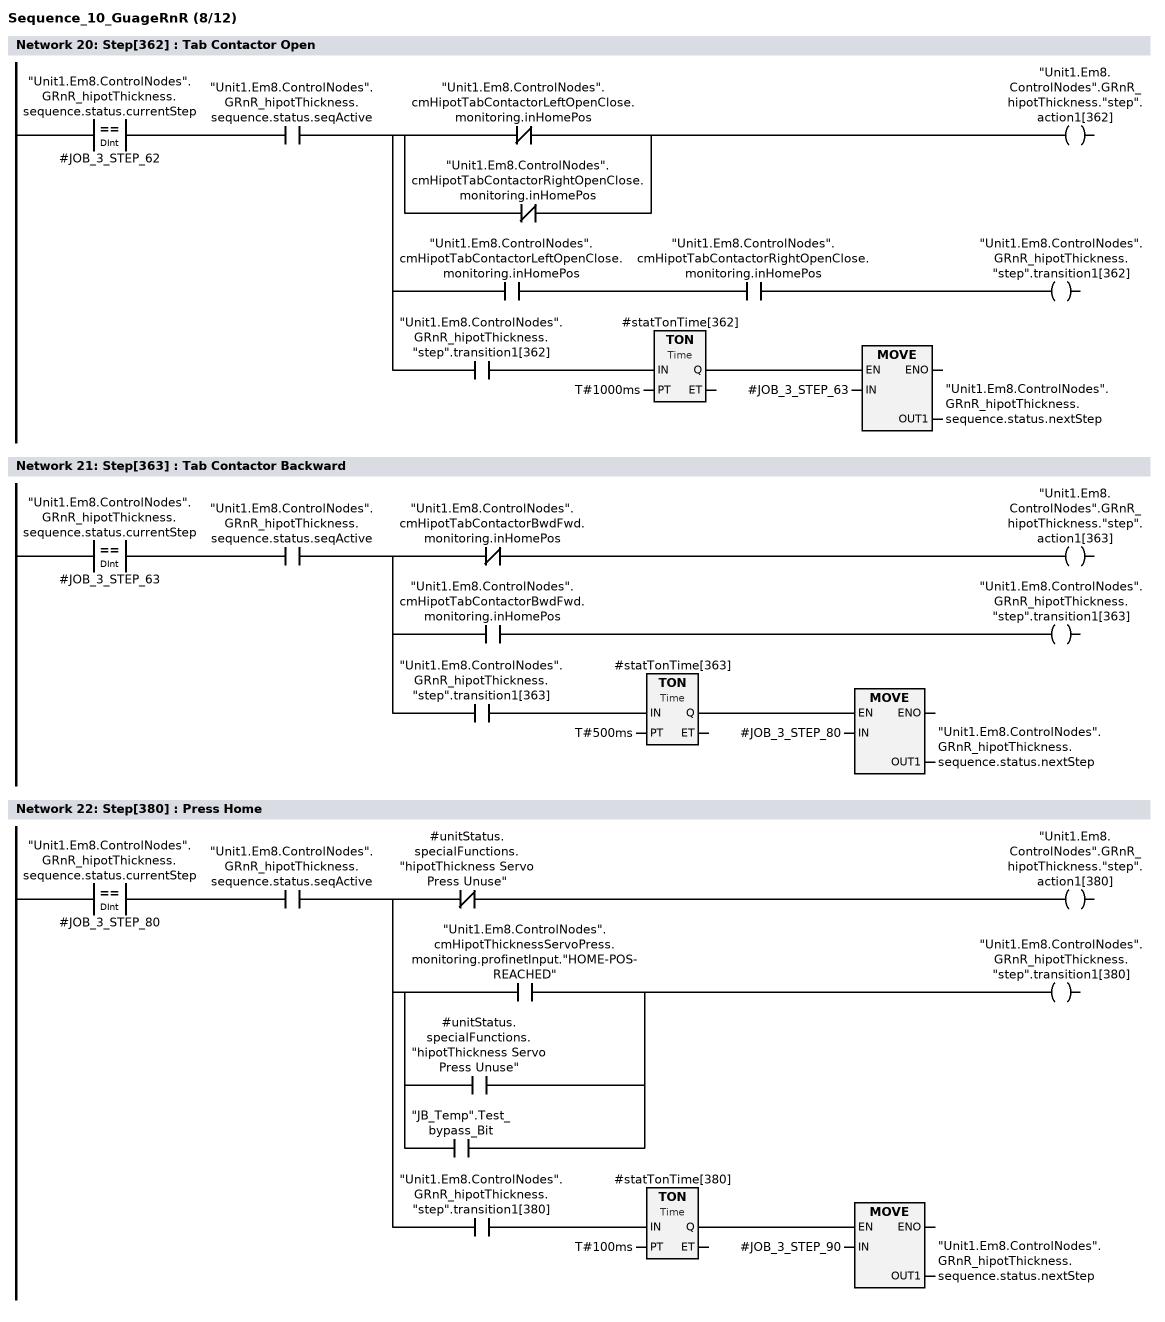
   RUNG wire#powerrail
      { S7_Templates := "SrcType := DInt" } EQ_Contact(in1 := "Unit1.Em8.ControlNodes".GRnR_hipotThickness.sequence.status.currentStep, in2 := #JOB_3_STEP_62)
      Contact( "Unit1.Em8.ControlNodes".GRnR_hipotThickness.sequence.status.seqActive )
      wire#w1
      I_Contact( "Unit1.Em8.ControlNodes".cmHipotTabContactorLeftOpenClose.monitoring.inHomePos )
      wire#w2
      Coil( "Unit1.Em8.ControlNodes".GRnR_hipotThickness."step".action1[362] )
   END_RUNG
   RUNG wire#w1
      I_Contact( "Unit1.Em8.ControlNodes".cmHipotTabContactorRightOpenClose.monitoring.inHomePos )
   END_RUNG wire#w2
   RUNG wire#w1
      Contact( "Unit1.Em8.ControlNodes".cmHipotTabContactorLeftOpenClose.monitoring.inHomePos )
      Contact( "Unit1.Em8.ControlNodes".cmHipotTabContactorRightOpenClose.monitoring.inHomePos )
      Coil( "Unit1.Em8.ControlNodes".GRnR_hipotThickness."step".transition1[362] )
   END_RUNG
   RUNG wire#w1
      Contact( "Unit1.Em8.ControlNodes".GRnR_hipotThickness."step".transition1[362] )
      { S7_Templates := "time_type := Time" } #statTonTime[362].TON(pt := T#1000ms, et =>)
      Move(in := #JOB_3_STEP_63, out1 => "Unit1.Em8.ControlNodes".GRnR_hipotThickness.sequence.status.nextStep)
   END_RUNG
   // the same network as SCL:
   #_w1 := ("Unit1.Em8.ControlNodes".GRnR_hipotThickness.sequence.status.currentStep = #JOB_3_STEP_62) AND "Unit1.Em8.ControlNodes".GRnR_hipotThickness.sequence.status.seqActive;
   "Unit1.Em8.ControlNodes".GRnR_hipotThickness."step".action1[362] := #_w1 AND (NOT "Unit1.Em8.ControlNodes".cmHipotTabContactorLeftOpenClose.monitoring.inHomePos OR NOT "Unit1.Em8.ControlNodes".cmHipotTabContactorRightOpenClose.monitoring.inHomePos);
   "Unit1.Em8.ControlNodes".GRnR_hipotThickness."step".transition1[362] := #_w1 AND "Unit1.Em8.ControlNodes".cmHipotTabContactorLeftOpenClose.monitoring.inHomePos AND "Unit1.Em8.ControlNodes".cmHipotTabContactorRightOpenClose.monitoring.inHomePos;
   #statTonTime[362].TON(IN := #_w1 AND "Unit1.Em8.ControlNodes".GRnR_hipotThickness."step".transition1[362],
                         PT := T#1000ms);
   IF #statTonTime[362].Q THEN
       "Unit1.Em8.ControlNodes".GRnR_hipotThickness.sequence.status.nextStep := #JOB_3_STEP_63;
   END_IF;
END_REGION

REGION Network 21: Step[363] : Tab Contactor Backward
   RUNG wire#powerrail
      { S7_Templates := "SrcType := DInt" } EQ_Contact(in1 := "Unit1.Em8.ControlNodes".GRnR_hipotThickness.sequence.status.currentStep, in2 := #JOB_3_STEP_63)
      Contact( "Unit1.Em8.ControlNodes".GRnR_hipotThickness.sequence.status.seqActive )
      wire#w1
      I_Contact( "Unit1.Em8.ControlNodes".cmHipotTabContactorBwdFwd.monitoring.inHomePos )
      Coil( "Unit1.Em8.ControlNodes".GRnR_hipotThickness."step".action1[363] )
   END_RUNG
   RUNG wire#w1
      Contact( "Unit1.Em8.ControlNodes".cmHipotTabContactorBwdFwd.monitoring.inHomePos )
      Coil( "Unit1.Em8.ControlNodes".GRnR_hipotThickness."step".transition1[363] )
   END_RUNG
   RUNG wire#w1
      Contact( "Unit1.Em8.ControlNodes".GRnR_hipotThickness."step".transition1[363] )
      { S7_Templates := "time_type := Time" } #statTonTime[363].TON(pt := T#500ms, et =>)
      Move(in := #JOB_3_STEP_80, out1 => "Unit1.Em8.ControlNodes".GRnR_hipotThickness.sequence.status.nextStep)
   END_RUNG
   // the same network as SCL:
   #_w1 := ("Unit1.Em8.ControlNodes".GRnR_hipotThickness.sequence.status.currentStep = #JOB_3_STEP_63) AND "Unit1.Em8.ControlNodes".GRnR_hipotThickness.sequence.status.seqActive;
   "Unit1.Em8.ControlNodes".GRnR_hipotThickness."step".action1[363] := #_w1 AND NOT "Unit1.Em8.ControlNodes".cmHipotTabContactorBwdFwd.monitoring.inHomePos;
   "Unit1.Em8.ControlNodes".GRnR_hipotThickness."step".transition1[363] := #_w1 AND "Unit1.Em8.ControlNodes".cmHipotTabContactorBwdFwd.monitoring.inHomePos;
   #statTonTime[363].TON(IN := #_w1 AND "Unit1.Em8.ControlNodes".GRnR_hipotThickness."step".transition1[363],
                         PT := T#500ms);
   IF #statTonTime[363].Q THEN
       "Unit1.Em8.ControlNodes".GRnR_hipotThickness.sequence.status.nextStep := #JOB_3_STEP_80;
   END_IF;
END_REGION

REGION Network 22: Step[380] : Press Home
   RUNG wire#powerrail
      { S7_Templates := "SrcType := DInt" } EQ_Contact(in1 := "Unit1.Em8.ControlNodes".GRnR_hipotThickness.sequence.status.currentStep, in2 := #JOB_3_STEP_80)
      Contact( "Unit1.Em8.ControlNodes".GRnR_hipotThickness.sequence.status.seqActive )
      wire#w1
      I_Contact( #unitStatus.specialFunctions."hipotThickness Servo Press Unuse" )
      Coil( "Unit1.Em8.ControlNodes".GRnR_hipotThickness."step".action1[380] )
   END_RUNG
   RUNG wire#w1
      Contact( "Unit1.Em8.ControlNodes".cmHipotThicknessServoPress.monitoring.profinetInput."HOME-POS-REACHED" )
      wire#w2
      Coil( "Unit1.Em8.ControlNodes".GRnR_hipotThickness."step".transition1[380] )
   END_RUNG
   RUNG wire#w1
      Contact( #unitStatus.specialFunctions."hipotThickness Servo Press Unuse" )
   END_RUNG wire#w2
   RUNG wire#w1
      Contact( "JB_Temp".Test_bypass_Bit )
   END_RUNG wire#w2
   RUNG wire#w1
      Contact( "Unit1.Em8.ControlNodes".GRnR_hipotThickness."step".transition1[380] )
      { S7_Templates := "time_type := Time" } #statTonTime[380].TON(pt := T#100ms, et =>)
      Move(in := #JOB_3_STEP_90, out1 => "Unit1.Em8.ControlNodes".GRnR_hipotThickness.sequence.status.nextStep)
   END_RUNG
   // the same network as SCL:
   #_w1 := ("Unit1.Em8.ControlNodes".GRnR_hipotThickness.sequence.status.currentStep = #JOB_3_STEP_80) AND "Unit1.Em8.ControlNodes".GRnR_hipotThickness.sequence.status.seqActive;
   "Unit1.Em8.ControlNodes".GRnR_hipotThickness."step".action1[380] := #_w1 AND NOT #unitStatus.specialFunctions."hipotThickness Servo Press Unuse";
   "Unit1.Em8.ControlNodes".GRnR_hipotThickness."step".transition1[380] := #_w1 AND ("Unit1.Em8.ControlNodes".cmHipotThicknessServoPress.monitoring.profinetInput."HOME-POS-REACHED" OR #unitStatus.specialFunctions."hipotThickness Servo Press Unuse" OR "JB_Temp".Test_bypass_Bit);
   #statTonTime[380].TON(IN := #_w1 AND "Unit1.Em8.ControlNodes".GRnR_hipotThickness."step".transition1[380],
                         PT := T#100ms);
   IF #statTonTime[380].Q THEN
       "Unit1.Em8.ControlNodes".GRnR_hipotThickness.sequence.status.nextStep := #JOB_3_STEP_90;
   END_IF;
END_REGION

REGION Network 23: Step[390] : JOB[3] Step End
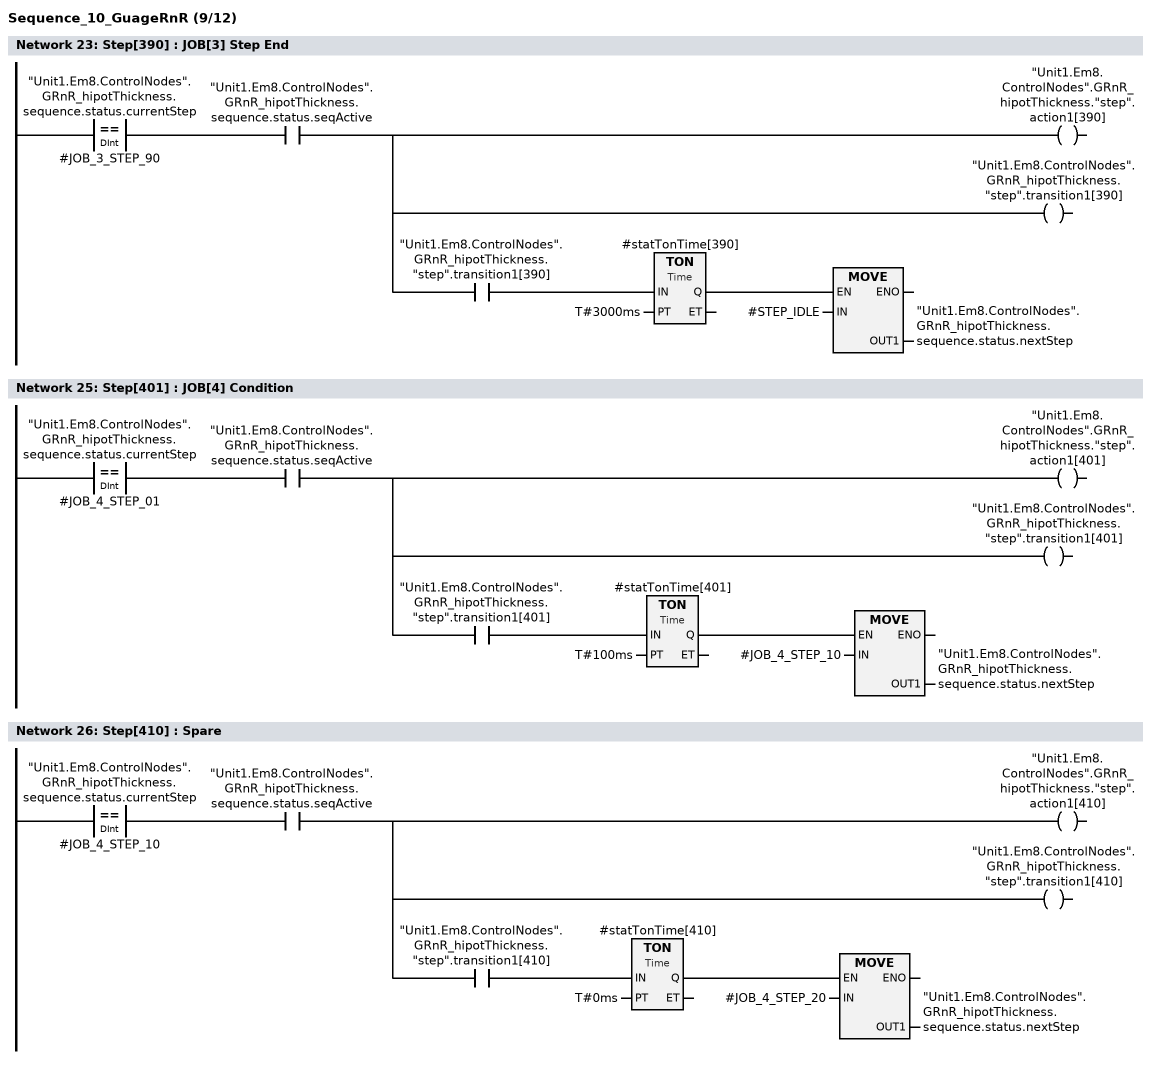
   RUNG wire#powerrail
      { S7_Templates := "SrcType := DInt" } EQ_Contact(in1 := "Unit1.Em8.ControlNodes".GRnR_hipotThickness.sequence.status.currentStep, in2 := #JOB_3_STEP_90)
      Contact( "Unit1.Em8.ControlNodes".GRnR_hipotThickness.sequence.status.seqActive )
      wire#w1
      Coil( "Unit1.Em8.ControlNodes".GRnR_hipotThickness."step".action1[390] )
   END_RUNG
   RUNG wire#w1
      Coil( "Unit1.Em8.ControlNodes".GRnR_hipotThickness."step".transition1[390] )
   END_RUNG
   RUNG wire#w1
      Contact( "Unit1.Em8.ControlNodes".GRnR_hipotThickness."step".transition1[390] )
      { S7_Templates := "time_type := Time" } #statTonTime[390].TON(pt := T#3000ms, et =>)
      Move(in := #STEP_IDLE, out1 => "Unit1.Em8.ControlNodes".GRnR_hipotThickness.sequence.status.nextStep)
   END_RUNG
   // the same network as SCL:
   "Unit1.Em8.ControlNodes".GRnR_hipotThickness."step".action1[390] := ("Unit1.Em8.ControlNodes".GRnR_hipotThickness.sequence.status.currentStep = #JOB_3_STEP_90) AND "Unit1.Em8.ControlNodes".GRnR_hipotThickness.sequence.status.seqActive;
   "Unit1.Em8.ControlNodes".GRnR_hipotThickness."step".transition1[390] := ("Unit1.Em8.ControlNodes".GRnR_hipotThickness.sequence.status.currentStep = #JOB_3_STEP_90) AND "Unit1.Em8.ControlNodes".GRnR_hipotThickness.sequence.status.seqActive;
   #statTonTime[390].TON(IN := ("Unit1.Em8.ControlNodes".GRnR_hipotThickness.sequence.status.currentStep = #JOB_3_STEP_90) AND "Unit1.Em8.ControlNodes".GRnR_hipotThickness.sequence.status.seqActive AND "Unit1.Em8.ControlNodes".GRnR_hipotThickness."step".transition1[390],
                         PT := T#3000ms);
   IF #statTonTime[390].Q THEN
       "Unit1.Em8.ControlNodes".GRnR_hipotThickness.sequence.status.nextStep := #STEP_IDLE;
   END_IF;
END_REGION

REGION Network 24: *************** JOB[4] JR PUT=AUTO ***********************
END_REGION

REGION Network 25: Step[401] : JOB[4] Condition
   RUNG wire#powerrail
      { S7_Templates := "SrcType := DInt" } EQ_Contact(in1 := "Unit1.Em8.ControlNodes".GRnR_hipotThickness.sequence.status.currentStep, in2 := #JOB_4_STEP_01)
      Contact( "Unit1.Em8.ControlNodes".GRnR_hipotThickness.sequence.status.seqActive )
      wire#w1
      Coil( "Unit1.Em8.ControlNodes".GRnR_hipotThickness."step".action1[401] )
   END_RUNG
   RUNG wire#w1
      Coil( "Unit1.Em8.ControlNodes".GRnR_hipotThickness."step".transition1[401] )
   END_RUNG
   RUNG wire#w1
      Contact( "Unit1.Em8.ControlNodes".GRnR_hipotThickness."step".transition1[401] )
      { S7_Templates := "time_type := Time" } #statTonTime[401].TON(pt := T#100ms, et =>)
      Move(in := #JOB_4_STEP_10, out1 => "Unit1.Em8.ControlNodes".GRnR_hipotThickness.sequence.status.nextStep)
   END_RUNG
   // the same network as SCL:
   "Unit1.Em8.ControlNodes".GRnR_hipotThickness."step".action1[401] := ("Unit1.Em8.ControlNodes".GRnR_hipotThickness.sequence.status.currentStep = #JOB_4_STEP_01) AND "Unit1.Em8.ControlNodes".GRnR_hipotThickness.sequence.status.seqActive;
   "Unit1.Em8.ControlNodes".GRnR_hipotThickness."step".transition1[401] := ("Unit1.Em8.ControlNodes".GRnR_hipotThickness.sequence.status.currentStep = #JOB_4_STEP_01) AND "Unit1.Em8.ControlNodes".GRnR_hipotThickness.sequence.status.seqActive;
   #statTonTime[401].TON(IN := ("Unit1.Em8.ControlNodes".GRnR_hipotThickness.sequence.status.currentStep = #JOB_4_STEP_01) AND "Unit1.Em8.ControlNodes".GRnR_hipotThickness.sequence.status.seqActive AND "Unit1.Em8.ControlNodes".GRnR_hipotThickness."step".transition1[401],
                         PT := T#100ms);
   IF #statTonTime[401].Q THEN
       "Unit1.Em8.ControlNodes".GRnR_hipotThickness.sequence.status.nextStep := #JOB_4_STEP_10;
   END_IF;
END_REGION

REGION Network 26: Step[410] : Spare
   RUNG wire#powerrail
      { S7_Templates := "SrcType := DInt" } EQ_Contact(in1 := "Unit1.Em8.ControlNodes".GRnR_hipotThickness.sequence.status.currentStep, in2 := #JOB_4_STEP_10)
      Contact( "Unit1.Em8.ControlNodes".GRnR_hipotThickness.sequence.status.seqActive )
      wire#w1
      Coil( "Unit1.Em8.ControlNodes".GRnR_hipotThickness."step".action1[410] )
   END_RUNG
   RUNG wire#w1
      Coil( "Unit1.Em8.ControlNodes".GRnR_hipotThickness."step".transition1[410] )
   END_RUNG
   RUNG wire#w1
      Contact( "Unit1.Em8.ControlNodes".GRnR_hipotThickness."step".transition1[410] )
      { S7_Templates := "time_type := Time" } #statTonTime[410].TON(pt := T#0ms, et =>)
      Move(in := #JOB_4_STEP_20, out1 => "Unit1.Em8.ControlNodes".GRnR_hipotThickness.sequence.status.nextStep)
   END_RUNG
   // the same network as SCL:
   "Unit1.Em8.ControlNodes".GRnR_hipotThickness."step".action1[410] := ("Unit1.Em8.ControlNodes".GRnR_hipotThickness.sequence.status.currentStep = #JOB_4_STEP_10) AND "Unit1.Em8.ControlNodes".GRnR_hipotThickness.sequence.status.seqActive;
   "Unit1.Em8.ControlNodes".GRnR_hipotThickness."step".transition1[410] := ("Unit1.Em8.ControlNodes".GRnR_hipotThickness.sequence.status.currentStep = #JOB_4_STEP_10) AND "Unit1.Em8.ControlNodes".GRnR_hipotThickness.sequence.status.seqActive;
   #statTonTime[410].TON(IN := ("Unit1.Em8.ControlNodes".GRnR_hipotThickness.sequence.status.currentStep = #JOB_4_STEP_10) AND "Unit1.Em8.ControlNodes".GRnR_hipotThickness.sequence.status.seqActive AND "Unit1.Em8.ControlNodes".GRnR_hipotThickness."step".transition1[410],
                         PT := T#0ms);
   IF #statTonTime[410].Q THEN
       "Unit1.Em8.ControlNodes".GRnR_hipotThickness.sequence.status.nextStep := #JOB_4_STEP_20;
   END_IF;
END_REGION

REGION Network 27: Step[420] : Stage Lift Up
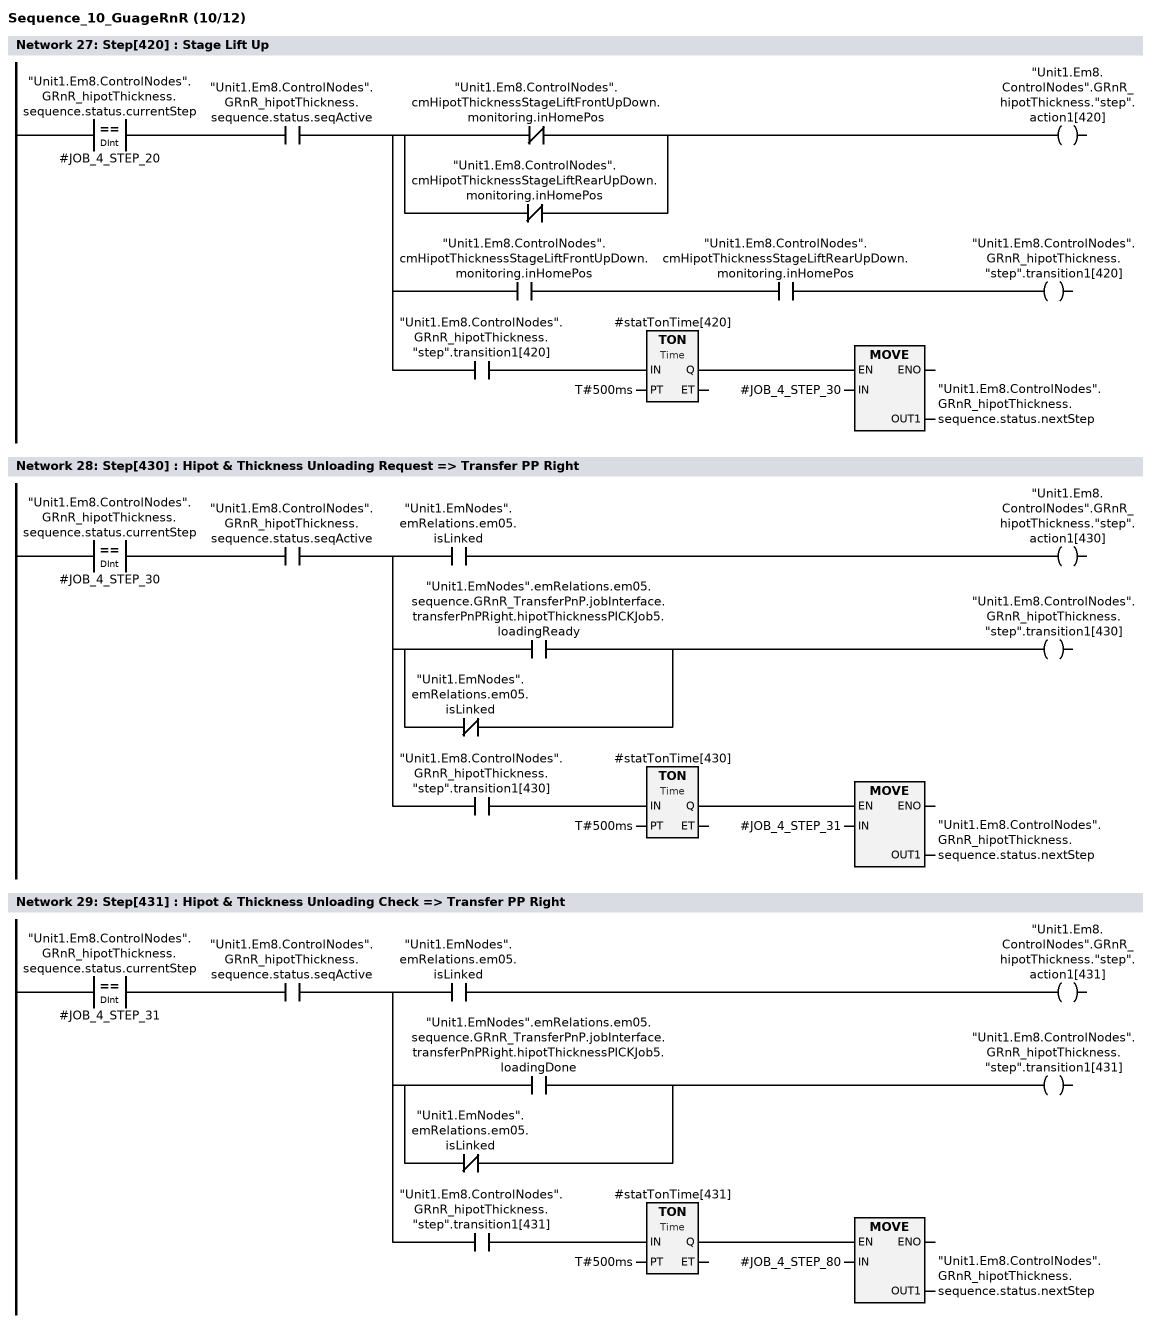
   RUNG wire#powerrail
      { S7_Templates := "SrcType := DInt" } EQ_Contact(in1 := "Unit1.Em8.ControlNodes".GRnR_hipotThickness.sequence.status.currentStep, in2 := #JOB_4_STEP_20)
      Contact( "Unit1.Em8.ControlNodes".GRnR_hipotThickness.sequence.status.seqActive )
      wire#w1
      I_Contact( "Unit1.Em8.ControlNodes".cmHipotThicknessStageLiftFrontUpDown.monitoring.inHomePos )
      wire#w2
      Coil( "Unit1.Em8.ControlNodes".GRnR_hipotThickness."step".action1[420] )
   END_RUNG
   RUNG wire#w1
      I_Contact( "Unit1.Em8.ControlNodes".cmHipotThicknessStageLiftRearUpDown.monitoring.inHomePos )
   END_RUNG wire#w2
   RUNG wire#w1
      Contact( "Unit1.Em8.ControlNodes".cmHipotThicknessStageLiftFrontUpDown.monitoring.inHomePos )
      Contact( "Unit1.Em8.ControlNodes".cmHipotThicknessStageLiftRearUpDown.monitoring.inHomePos )
      Coil( "Unit1.Em8.ControlNodes".GRnR_hipotThickness."step".transition1[420] )
   END_RUNG
   RUNG wire#w1
      Contact( "Unit1.Em8.ControlNodes".GRnR_hipotThickness."step".transition1[420] )
      { S7_Templates := "time_type := Time" } #statTonTime[420].TON(pt := T#500ms, et =>)
      Move(in := #JOB_4_STEP_30, out1 => "Unit1.Em8.ControlNodes".GRnR_hipotThickness.sequence.status.nextStep)
   END_RUNG
   // the same network as SCL:
   #_w1 := ("Unit1.Em8.ControlNodes".GRnR_hipotThickness.sequence.status.currentStep = #JOB_4_STEP_20) AND "Unit1.Em8.ControlNodes".GRnR_hipotThickness.sequence.status.seqActive;
   "Unit1.Em8.ControlNodes".GRnR_hipotThickness."step".action1[420] := #_w1 AND (NOT "Unit1.Em8.ControlNodes".cmHipotThicknessStageLiftFrontUpDown.monitoring.inHomePos OR NOT "Unit1.Em8.ControlNodes".cmHipotThicknessStageLiftRearUpDown.monitoring.inHomePos);
   "Unit1.Em8.ControlNodes".GRnR_hipotThickness."step".transition1[420] := #_w1 AND "Unit1.Em8.ControlNodes".cmHipotThicknessStageLiftFrontUpDown.monitoring.inHomePos AND "Unit1.Em8.ControlNodes".cmHipotThicknessStageLiftRearUpDown.monitoring.inHomePos;
   #statTonTime[420].TON(IN := #_w1 AND "Unit1.Em8.ControlNodes".GRnR_hipotThickness."step".transition1[420],
                         PT := T#500ms);
   IF #statTonTime[420].Q THEN
       "Unit1.Em8.ControlNodes".GRnR_hipotThickness.sequence.status.nextStep := #JOB_4_STEP_30;
   END_IF;
END_REGION

REGION Network 28: Step[430] : Hipot & Thickness Unloading Request => Transfer PP Right
   RUNG wire#powerrail
      { S7_Templates := "SrcType := DInt" } EQ_Contact(in1 := "Unit1.Em8.ControlNodes".GRnR_hipotThickness.sequence.status.currentStep, in2 := #JOB_4_STEP_30)
      Contact( "Unit1.Em8.ControlNodes".GRnR_hipotThickness.sequence.status.seqActive )
      wire#w1
      Contact( "Unit1.EmNodes".emRelations.em05.isLinked )
      Coil( "Unit1.Em8.ControlNodes".GRnR_hipotThickness."step".action1[430] )
   END_RUNG
   RUNG wire#w1
      Contact( "Unit1.EmNodes".emRelations.em05.sequence.GRnR_TransferPnP.jobInterface.transferPnPRight.hipotThicknessPICKJob5.loadingReady )
      wire#w2
      Coil( "Unit1.Em8.ControlNodes".GRnR_hipotThickness."step".transition1[430] )
   END_RUNG
   RUNG wire#w1
      I_Contact( "Unit1.EmNodes".emRelations.em05.isLinked )
   END_RUNG wire#w2
   RUNG wire#w1
      Contact( "Unit1.Em8.ControlNodes".GRnR_hipotThickness."step".transition1[430] )
      { S7_Templates := "time_type := Time" } #statTonTime[430].TON(pt := T#500ms, et =>)
      Move(in := #JOB_4_STEP_31, out1 => "Unit1.Em8.ControlNodes".GRnR_hipotThickness.sequence.status.nextStep)
   END_RUNG
   // the same network as SCL:
   #_w1 := ("Unit1.Em8.ControlNodes".GRnR_hipotThickness.sequence.status.currentStep = #JOB_4_STEP_30) AND "Unit1.Em8.ControlNodes".GRnR_hipotThickness.sequence.status.seqActive;
   "Unit1.Em8.ControlNodes".GRnR_hipotThickness."step".action1[430] := #_w1 AND "Unit1.EmNodes".emRelations.em05.isLinked;
   "Unit1.Em8.ControlNodes".GRnR_hipotThickness."step".transition1[430] := #_w1 AND ("Unit1.EmNodes".emRelations.em05.sequence.GRnR_TransferPnP.jobInterface.transferPnPRight.hipotThicknessPICKJob5.loadingReady OR NOT "Unit1.EmNodes".emRelations.em05.isLinked);
   #statTonTime[430].TON(IN := #_w1 AND "Unit1.Em8.ControlNodes".GRnR_hipotThickness."step".transition1[430],
                         PT := T#500ms);
   IF #statTonTime[430].Q THEN
       "Unit1.Em8.ControlNodes".GRnR_hipotThickness.sequence.status.nextStep := #JOB_4_STEP_31;
   END_IF;
END_REGION

REGION Network 29: Step[431] : Hipot & Thickness Unloading Check => Transfer PP Right
   RUNG wire#powerrail
      { S7_Templates := "SrcType := DInt" } EQ_Contact(in1 := "Unit1.Em8.ControlNodes".GRnR_hipotThickness.sequence.status.currentStep, in2 := #JOB_4_STEP_31)
      Contact( "Unit1.Em8.ControlNodes".GRnR_hipotThickness.sequence.status.seqActive )
      wire#w1
      Contact( "Unit1.EmNodes".emRelations.em05.isLinked )
      Coil( "Unit1.Em8.ControlNodes".GRnR_hipotThickness."step".action1[431] )
   END_RUNG
   RUNG wire#w1
      Contact( "Unit1.EmNodes".emRelations.em05.sequence.GRnR_TransferPnP.jobInterface.transferPnPRight.hipotThicknessPICKJob5.loadingDone )
      wire#w2
      Coil( "Unit1.Em8.ControlNodes".GRnR_hipotThickness."step".transition1[431] )
   END_RUNG
   RUNG wire#w1
      I_Contact( "Unit1.EmNodes".emRelations.em05.isLinked )
   END_RUNG wire#w2
   RUNG wire#w1
      Contact( "Unit1.Em8.ControlNodes".GRnR_hipotThickness."step".transition1[431] )
      { S7_Templates := "time_type := Time" } #statTonTime[431].TON(pt := T#500ms, et =>)
      Move(in := #JOB_4_STEP_80, out1 => "Unit1.Em8.ControlNodes".GRnR_hipotThickness.sequence.status.nextStep)
   END_RUNG
   // the same network as SCL:
   #_w1 := ("Unit1.Em8.ControlNodes".GRnR_hipotThickness.sequence.status.currentStep = #JOB_4_STEP_31) AND "Unit1.Em8.ControlNodes".GRnR_hipotThickness.sequence.status.seqActive;
   "Unit1.Em8.ControlNodes".GRnR_hipotThickness."step".action1[431] := #_w1 AND "Unit1.EmNodes".emRelations.em05.isLinked;
   "Unit1.Em8.ControlNodes".GRnR_hipotThickness."step".transition1[431] := #_w1 AND ("Unit1.EmNodes".emRelations.em05.sequence.GRnR_TransferPnP.jobInterface.transferPnPRight.hipotThicknessPICKJob5.loadingDone OR NOT "Unit1.EmNodes".emRelations.em05.isLinked);
   #statTonTime[431].TON(IN := #_w1 AND "Unit1.Em8.ControlNodes".GRnR_hipotThickness."step".transition1[431],
                         PT := T#500ms);
   IF #statTonTime[431].Q THEN
       "Unit1.Em8.ControlNodes".GRnR_hipotThickness.sequence.status.nextStep := #JOB_4_STEP_80;
   END_IF;
END_REGION

REGION Network 30: Step[480] : Stage Lift Down
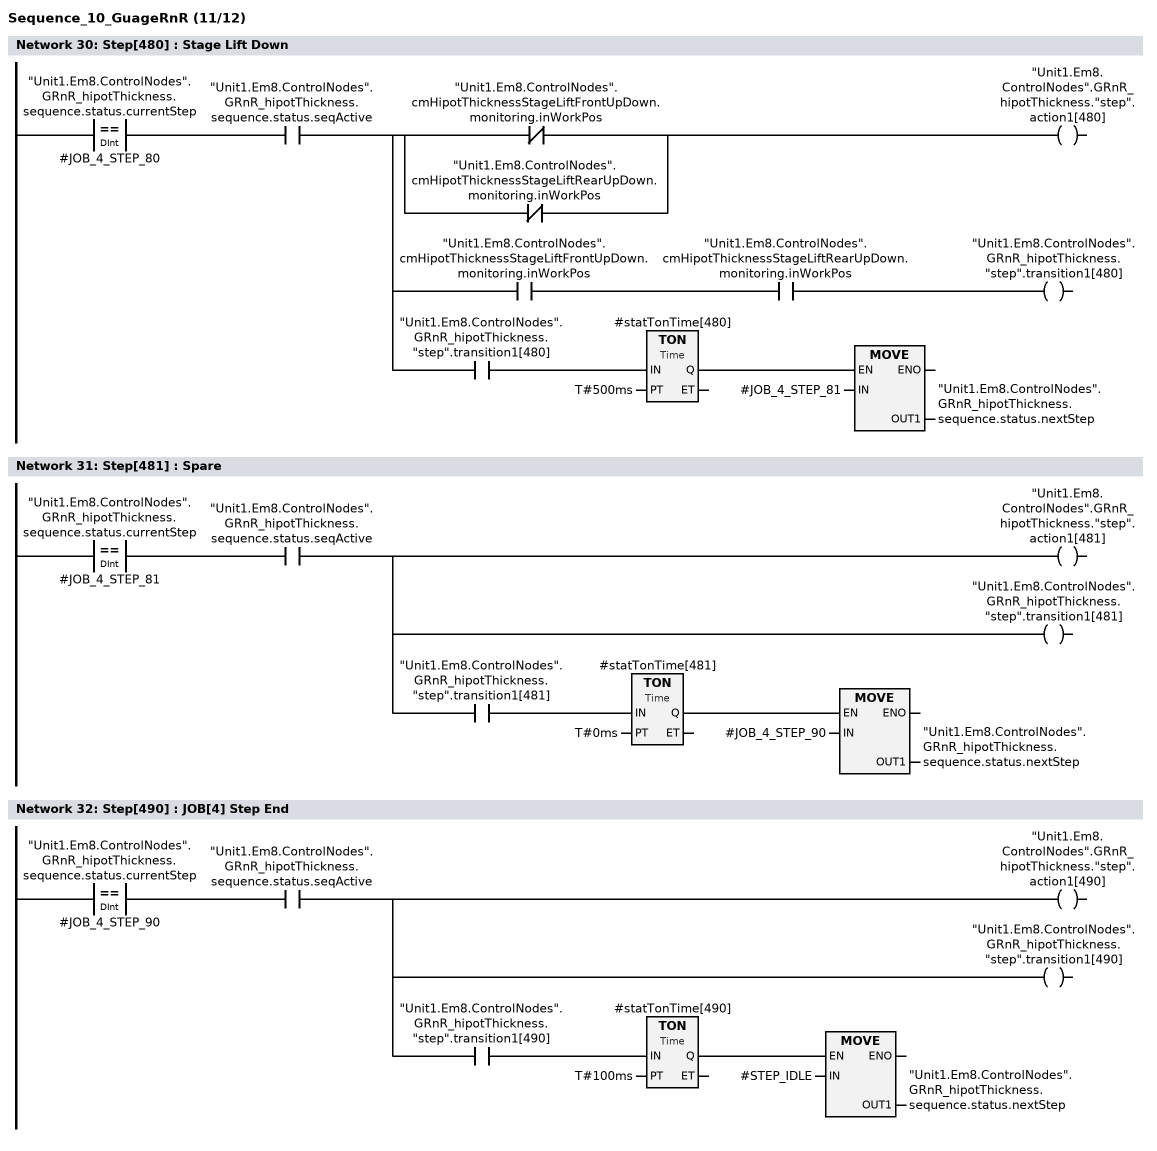
   RUNG wire#powerrail
      { S7_Templates := "SrcType := DInt" } EQ_Contact(in1 := "Unit1.Em8.ControlNodes".GRnR_hipotThickness.sequence.status.currentStep, in2 := #JOB_4_STEP_80)
      Contact( "Unit1.Em8.ControlNodes".GRnR_hipotThickness.sequence.status.seqActive )
      wire#w1
      I_Contact( "Unit1.Em8.ControlNodes".cmHipotThicknessStageLiftFrontUpDown.monitoring.inWorkPos )
      wire#w2
      Coil( "Unit1.Em8.ControlNodes".GRnR_hipotThickness."step".action1[480] )
   END_RUNG
   RUNG wire#w1
      I_Contact( "Unit1.Em8.ControlNodes".cmHipotThicknessStageLiftRearUpDown.monitoring.inWorkPos )
   END_RUNG wire#w2
   RUNG wire#w1
      Contact( "Unit1.Em8.ControlNodes".cmHipotThicknessStageLiftFrontUpDown.monitoring.inWorkPos )
      Contact( "Unit1.Em8.ControlNodes".cmHipotThicknessStageLiftRearUpDown.monitoring.inWorkPos )
      Coil( "Unit1.Em8.ControlNodes".GRnR_hipotThickness."step".transition1[480] )
   END_RUNG
   RUNG wire#w1
      Contact( "Unit1.Em8.ControlNodes".GRnR_hipotThickness."step".transition1[480] )
      { S7_Templates := "time_type := Time" } #statTonTime[480].TON(pt := T#500ms, et =>)
      Move(in := #JOB_4_STEP_81, out1 => "Unit1.Em8.ControlNodes".GRnR_hipotThickness.sequence.status.nextStep)
   END_RUNG
   // the same network as SCL:
   #_w1 := ("Unit1.Em8.ControlNodes".GRnR_hipotThickness.sequence.status.currentStep = #JOB_4_STEP_80) AND "Unit1.Em8.ControlNodes".GRnR_hipotThickness.sequence.status.seqActive;
   "Unit1.Em8.ControlNodes".GRnR_hipotThickness."step".action1[480] := #_w1 AND (NOT "Unit1.Em8.ControlNodes".cmHipotThicknessStageLiftFrontUpDown.monitoring.inWorkPos OR NOT "Unit1.Em8.ControlNodes".cmHipotThicknessStageLiftRearUpDown.monitoring.inWorkPos);
   "Unit1.Em8.ControlNodes".GRnR_hipotThickness."step".transition1[480] := #_w1 AND "Unit1.Em8.ControlNodes".cmHipotThicknessStageLiftFrontUpDown.monitoring.inWorkPos AND "Unit1.Em8.ControlNodes".cmHipotThicknessStageLiftRearUpDown.monitoring.inWorkPos;
   #statTonTime[480].TON(IN := #_w1 AND "Unit1.Em8.ControlNodes".GRnR_hipotThickness."step".transition1[480],
                         PT := T#500ms);
   IF #statTonTime[480].Q THEN
       "Unit1.Em8.ControlNodes".GRnR_hipotThickness.sequence.status.nextStep := #JOB_4_STEP_81;
   END_IF;
END_REGION

REGION Network 31: Step[481] : Spare
   RUNG wire#powerrail
      { S7_Templates := "SrcType := DInt" } EQ_Contact(in1 := "Unit1.Em8.ControlNodes".GRnR_hipotThickness.sequence.status.currentStep, in2 := #JOB_4_STEP_81)
      Contact( "Unit1.Em8.ControlNodes".GRnR_hipotThickness.sequence.status.seqActive )
      wire#w1
      Coil( "Unit1.Em8.ControlNodes".GRnR_hipotThickness."step".action1[481] )
   END_RUNG
   RUNG wire#w1
      Coil( "Unit1.Em8.ControlNodes".GRnR_hipotThickness."step".transition1[481] )
   END_RUNG
   RUNG wire#w1
      Contact( "Unit1.Em8.ControlNodes".GRnR_hipotThickness."step".transition1[481] )
      { S7_Templates := "time_type := Time" } #statTonTime[481].TON(pt := T#0ms, et =>)
      Move(in := #JOB_4_STEP_90, out1 => "Unit1.Em8.ControlNodes".GRnR_hipotThickness.sequence.status.nextStep)
   END_RUNG
   // the same network as SCL:
   "Unit1.Em8.ControlNodes".GRnR_hipotThickness."step".action1[481] := ("Unit1.Em8.ControlNodes".GRnR_hipotThickness.sequence.status.currentStep = #JOB_4_STEP_81) AND "Unit1.Em8.ControlNodes".GRnR_hipotThickness.sequence.status.seqActive;
   "Unit1.Em8.ControlNodes".GRnR_hipotThickness."step".transition1[481] := ("Unit1.Em8.ControlNodes".GRnR_hipotThickness.sequence.status.currentStep = #JOB_4_STEP_81) AND "Unit1.Em8.ControlNodes".GRnR_hipotThickness.sequence.status.seqActive;
   #statTonTime[481].TON(IN := ("Unit1.Em8.ControlNodes".GRnR_hipotThickness.sequence.status.currentStep = #JOB_4_STEP_81) AND "Unit1.Em8.ControlNodes".GRnR_hipotThickness.sequence.status.seqActive AND "Unit1.Em8.ControlNodes".GRnR_hipotThickness."step".transition1[481],
                         PT := T#0ms);
   IF #statTonTime[481].Q THEN
       "Unit1.Em8.ControlNodes".GRnR_hipotThickness.sequence.status.nextStep := #JOB_4_STEP_90;
   END_IF;
END_REGION

REGION Network 32: Step[490] : JOB[4] Step End
   RUNG wire#powerrail
      { S7_Templates := "SrcType := DInt" } EQ_Contact(in1 := "Unit1.Em8.ControlNodes".GRnR_hipotThickness.sequence.status.currentStep, in2 := #JOB_4_STEP_90)
      Contact( "Unit1.Em8.ControlNodes".GRnR_hipotThickness.sequence.status.seqActive )
      wire#w1
      Coil( "Unit1.Em8.ControlNodes".GRnR_hipotThickness."step".action1[490] )
   END_RUNG
   RUNG wire#w1
      Coil( "Unit1.Em8.ControlNodes".GRnR_hipotThickness."step".transition1[490] )
   END_RUNG
   RUNG wire#w1
      Contact( "Unit1.Em8.ControlNodes".GRnR_hipotThickness."step".transition1[490] )
      { S7_Templates := "time_type := Time" } #statTonTime[490].TON(pt := T#100ms, et =>)
      Move(in := #STEP_IDLE, out1 => "Unit1.Em8.ControlNodes".GRnR_hipotThickness.sequence.status.nextStep)
   END_RUNG
   // the same network as SCL:
   "Unit1.Em8.ControlNodes".GRnR_hipotThickness."step".action1[490] := ("Unit1.Em8.ControlNodes".GRnR_hipotThickness.sequence.status.currentStep = #JOB_4_STEP_90) AND "Unit1.Em8.ControlNodes".GRnR_hipotThickness.sequence.status.seqActive;
   "Unit1.Em8.ControlNodes".GRnR_hipotThickness."step".transition1[490] := ("Unit1.Em8.ControlNodes".GRnR_hipotThickness.sequence.status.currentStep = #JOB_4_STEP_90) AND "Unit1.Em8.ControlNodes".GRnR_hipotThickness.sequence.status.seqActive;
   #statTonTime[490].TON(IN := ("Unit1.Em8.ControlNodes".GRnR_hipotThickness.sequence.status.currentStep = #JOB_4_STEP_90) AND "Unit1.Em8.ControlNodes".GRnR_hipotThickness.sequence.status.seqActive AND "Unit1.Em8.ControlNodes".GRnR_hipotThickness."step".transition1[490],
                         PT := T#100ms);
   IF #statTonTime[490].Q THEN
       "Unit1.Em8.ControlNodes".GRnR_hipotThickness.sequence.status.nextStep := #STEP_IDLE;
   END_IF;
END_REGION

REGION Network 33: ******************** IMMEDIATE STOP *********************
END_REGION

REGION Network 34: Immediate Stop
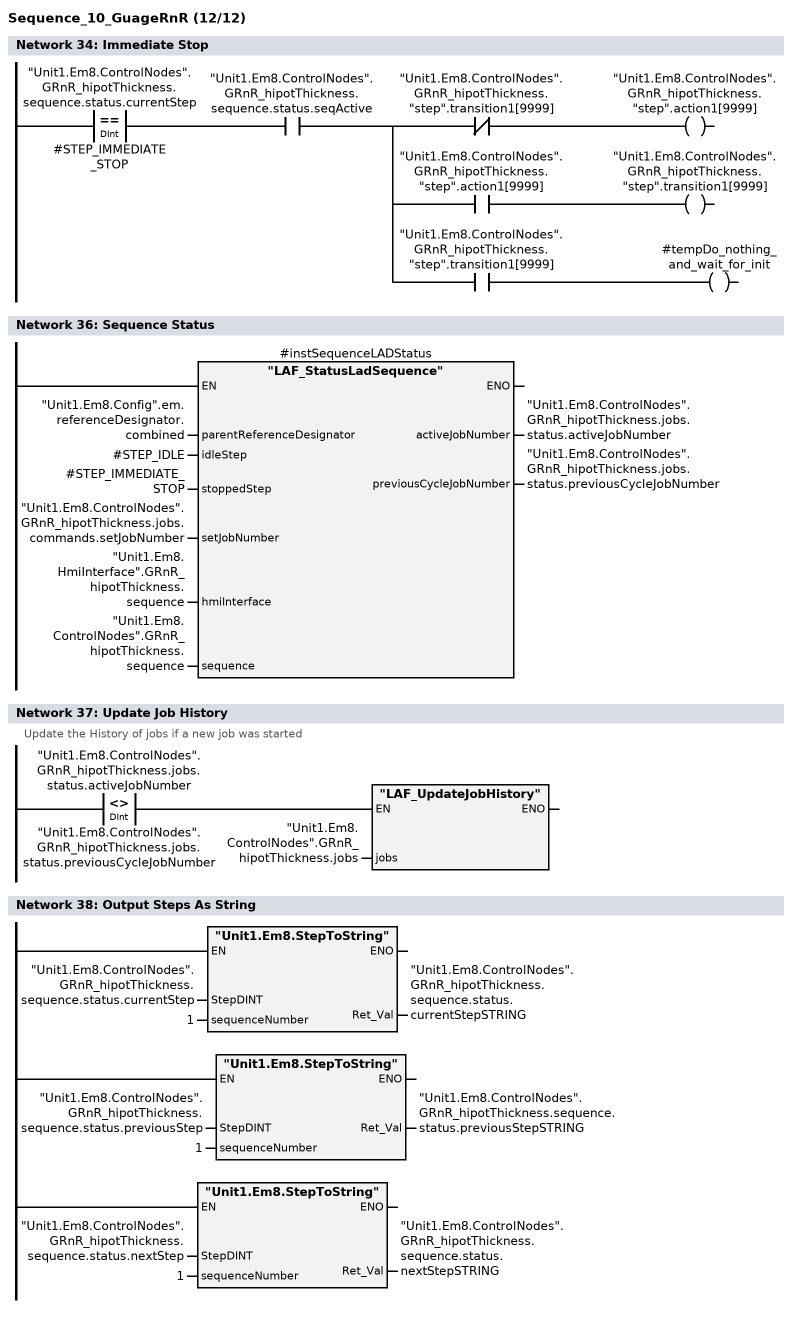
   RUNG wire#powerrail
      { S7_Templates := "SrcType := DInt" } EQ_Contact(in1 := "Unit1.Em8.ControlNodes".GRnR_hipotThickness.sequence.status.currentStep, in2 := #STEP_IMMEDIATE_STOP)
      Contact( "Unit1.Em8.ControlNodes".GRnR_hipotThickness.sequence.status.seqActive )
      wire#w1
      I_Contact( "Unit1.Em8.ControlNodes".GRnR_hipotThickness."step".transition1[9999] )
      Coil( "Unit1.Em8.ControlNodes".GRnR_hipotThickness."step".action1[9999] )
   END_RUNG
   RUNG wire#w1
      Contact( "Unit1.Em8.ControlNodes".GRnR_hipotThickness."step".action1[9999] )
      Coil( "Unit1.Em8.ControlNodes".GRnR_hipotThickness."step".transition1[9999] )
   END_RUNG
   RUNG wire#w1
      Contact( "Unit1.Em8.ControlNodes".GRnR_hipotThickness."step".transition1[9999] )
      Coil( #tempDo_nothing_and_wait_for_init )
   END_RUNG
   // the same network as SCL:
   #_w1 := ("Unit1.Em8.ControlNodes".GRnR_hipotThickness.sequence.status.currentStep = #STEP_IMMEDIATE_STOP) AND "Unit1.Em8.ControlNodes".GRnR_hipotThickness.sequence.status.seqActive;
   "Unit1.Em8.ControlNodes".GRnR_hipotThickness."step".action1[9999] := #_w1 AND NOT "Unit1.Em8.ControlNodes".GRnR_hipotThickness."step".transition1[9999];
   "Unit1.Em8.ControlNodes".GRnR_hipotThickness."step".transition1[9999] := #_w1 AND "Unit1.Em8.ControlNodes".GRnR_hipotThickness."step".action1[9999];
   #tempDo_nothing_and_wait_for_init := #_w1 AND "Unit1.Em8.ControlNodes".GRnR_hipotThickness."step".transition1[9999];
END_REGION

REGION Network 35: ********************** STATUS **************************
END_REGION

REGION Network 36: Sequence Status
   RUNG wire#powerrail
      #instSequenceLADStatus(parentReferenceDesignator := "Unit1.Em8.Config".em.referenceDesignator.combined, idleStep := #STEP_IDLE, stoppedStep := #STEP_IMMEDIATE_STOP, setJobNumber := "Unit1.Em8.ControlNodes".GRnR_hipotThickness.jobs.commands.setJobNumber, hmiInterface := "Unit1.Em8.HmiInterface".GRnR_hipotThickness.sequence, sequence := "Unit1.Em8.ControlNodes".GRnR_hipotThickness.sequence, activeJobNumber => "Unit1.Em8.ControlNodes".GRnR_hipotThickness.jobs.status.activeJobNumber, previousCycleJobNumber => "Unit1.Em8.ControlNodes".GRnR_hipotThickness.jobs.status.previousCycleJobNumber)
   END_RUNG
   // the same network as SCL:
   #instSequenceLADStatus(parentReferenceDesignator := "Unit1.Em8.Config".em.referenceDesignator.combined,   // "LAF_StatusLadSequence"
                          idleStep := #STEP_IDLE,
                          stoppedStep := #STEP_IMMEDIATE_STOP,
                          setJobNumber := "Unit1.Em8.ControlNodes".GRnR_hipotThickness.jobs.commands.setJobNumber,
                          hmiInterface := "Unit1.Em8.HmiInterface".GRnR_hipotThickness.sequence,
                          sequence := "Unit1.Em8.ControlNodes".GRnR_hipotThickness.sequence,
                          activeJobNumber => "Unit1.Em8.ControlNodes".GRnR_hipotThickness.jobs.status.activeJobNumber,
                          previousCycleJobNumber => "Unit1.Em8.ControlNodes".GRnR_hipotThickness.jobs.status.previousCycleJobNumber);
END_REGION

REGION Network 37: Update Job History
   // Update the History of jobs if a new job was started
   RUNG wire#powerrail
      { S7_Templates := "SrcType := DInt" } NE_Contact(in1 := "Unit1.Em8.ControlNodes".GRnR_hipotThickness.jobs.status.activeJobNumber, in2 := "Unit1.Em8.ControlNodes".GRnR_hipotThickness.jobs.status.previousCycleJobNumber)
      "LAF_UpdateJobHistory"(jobs := "Unit1.Em8.ControlNodes".GRnR_hipotThickness.jobs)
   END_RUNG
   // the same network as SCL:
   IF "Unit1.Em8.ControlNodes".GRnR_hipotThickness.jobs.status.activeJobNumber <> "Unit1.Em8.ControlNodes".GRnR_hipotThickness.jobs.status.previousCycleJobNumber THEN
       "LAF_UpdateJobHistory"(jobs := "Unit1.Em8.ControlNodes".GRnR_hipotThickness.jobs);
   END_IF;
END_REGION

REGION Network 38: Output Steps As String
   RUNG wire#powerrail
      "Unit1.Em8.StepToString"(StepDINT := "Unit1.Em8.ControlNodes".GRnR_hipotThickness.sequence.status.currentStep, sequenceNumber := 1, Ret_Val => "Unit1.Em8.ControlNodes".GRnR_hipotThickness.sequence.status.currentStepSTRING)
   END_RUNG
   RUNG wire#powerrail
      "Unit1.Em8.StepToString"(StepDINT := "Unit1.Em8.ControlNodes".GRnR_hipotThickness.sequence.status.previousStep, sequenceNumber := 1, Ret_Val => "Unit1.Em8.ControlNodes".GRnR_hipotThickness.sequence.status.previousStepSTRING)
   END_RUNG
   RUNG wire#powerrail
      "Unit1.Em8.StepToString"(StepDINT := "Unit1.Em8.ControlNodes".GRnR_hipotThickness.sequence.status.nextStep, sequenceNumber := 1, Ret_Val => "Unit1.Em8.ControlNodes".GRnR_hipotThickness.sequence.status.nextStepSTRING)
   END_RUNG
   // the same network as SCL:
   "Unit1.Em8.ControlNodes".GRnR_hipotThickness.sequence.status.currentStepSTRING := "Unit1.Em8.StepToString"(StepDINT := "Unit1.Em8.ControlNodes".GRnR_hipotThickness.sequence.status.currentStep,
                           sequenceNumber := 1);
   "Unit1.Em8.ControlNodes".GRnR_hipotThickness.sequence.status.previousStepSTRING := "Unit1.Em8.StepToString"(StepDINT := "Unit1.Em8.ControlNodes".GRnR_hipotThickness.sequence.status.previousStep,
                           sequenceNumber := 1);
   "Unit1.Em8.ControlNodes".GRnR_hipotThickness.sequence.status.nextStepSTRING := "Unit1.Em8.StepToString"(StepDINT := "Unit1.Em8.ControlNodes".GRnR_hipotThickness.sequence.status.nextStep,
                           sequenceNumber := 1);
END_REGION
END_FUNCTION_BLOCK
